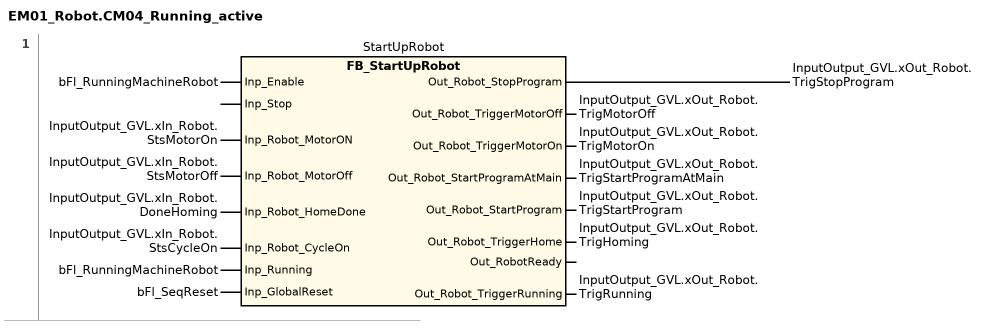
// NETWORK 1
StartUpRobot(
    Inp_Enable := bFl_RunningMachineRobot,
    Inp_Robot_MotorON := InputOutput_GVL.xIn_Robot.StsMotorOn,
    Inp_Robot_MotorOff := InputOutput_GVL.xIn_Robot.StsMotorOff,
    Inp_Robot_HomeDone := InputOutput_GVL.xIn_Robot.DoneHoming,
    Inp_Robot_CycleOn := InputOutput_GVL.xIn_Robot.StsCycleOn,
    Inp_Running := bFl_RunningMachineRobot,
    Inp_GlobalReset := bFl_SeqReset,
    Out_Robot_TriggerMotorOff => InputOutput_GVL.xOut_Robot.TrigMotorOff,
    Out_Robot_TriggerMotorOn => InputOutput_GVL.xOut_Robot.TrigMotorOn,
    Out_Robot_StartProgramAtMain => InputOutput_GVL.xOut_Robot.TrigStartProgramAtMain,
    Out_Robot_StartProgram => InputOutput_GVL.xOut_Robot.TrigStartProgram,
    Out_Robot_TriggerHome => InputOutput_GVL.xOut_Robot.TrigHoming,
    Out_Robot_TriggerRunning => InputOutput_GVL.xOut_Robot.TrigRunning); // FB_StartUpRobot
InputOutput_GVL.xOut_Robot.TrigStopProgram := StartUpRobot.Out_Robot_StopProgram;
END_ACTION

ACTION UP01_Backbone_active:
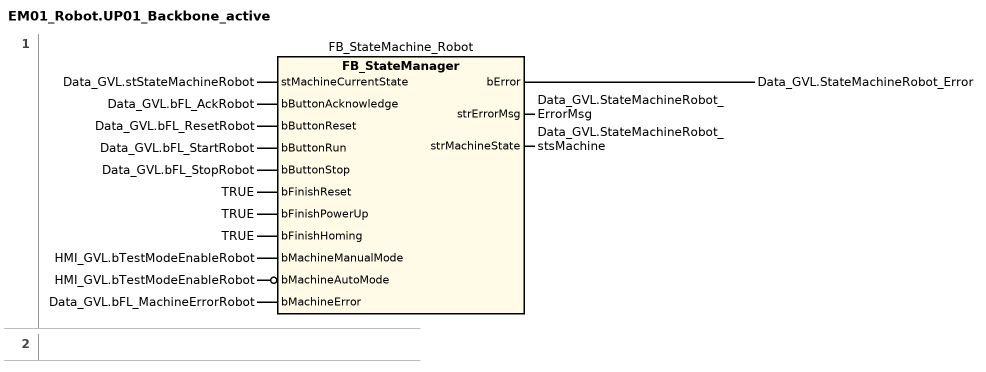
// NETWORK 1
FB_StateMachine_Robot(
    stMachineCurrentState := Data_GVL.stStateMachineRobot,
    bButtonAcknowledge := Data_GVL.bFL_AckRobot,
    bButtonReset := Data_GVL.bFL_ResetRobot,
    bButtonRun := Data_GVL.bFL_StartRobot,
    bButtonStop := Data_GVL.bFL_StopRobot,
    bFinishReset := TRUE,
    bFinishPowerUp := TRUE,
    bFinishHoming := TRUE,
    bMachineManualMode := HMI_GVL.bTestModeEnableRobot,
    bMachineAutoMode := NOT HMI_GVL.bTestModeEnableRobot,
    bMachineError := Data_GVL.bFL_MachineErrorRobot,
    strErrorMsg => Data_GVL.StateMachineRobot_ErrorMsg,
    strMachineState => Data_GVL.StateMachineRobot_stsMachine); // FB_StateManager
Data_GVL.StateMachineRobot_Error := FB_StateMachine_Robot.bError;

// NETWORK 2
END_ACTION

END_PROGRAM

// ---- POUs/Function_Block/General/FB_StateManager.TcPOU
FUNCTION_BLOCK FB_StateManager
VAR_IN_OUT
	stMachineCurrentState			: stMachineState;
END_VAR
VAR_INPUT
	bButtonAcknowledge				: BOOL;		// User Input for Error Acknowledgement
	bButtonReset					: BOOL;		// User Input for Reset 
	bButtonRun						: BOOL;		// User Input for Starting Machine Running Sequence
	bButtonStop						: BOOL;		// User Input for Stopping Machine Running Sequence
	bFinishReset					: BOOL;
	bFinishPowerUp					: BOOL;
	bFinishHoming					: BOOL;
	bMachineManualMode				: BOOL;		// Input(s) Required to Change Machine Operation Mode Into Manual Mode
	bMachineAutoMode				: BOOL;		// Input(s) Required to Change Machine Operation Mode Into Auto Mode
	bMachineError					: BOOL;		// Input(s) required to make the machine goes into error state
END_VAR
VAR_OUTPUT
	bError							: BOOL;		
	strErrorMsg						: STRING;	
	strMachineState					: STRING;
END_VAR
VAR
	bFL_AutoModeActive				: BOOL;
	bFL_ManualModeActive			: BOOL;
	bInit							: BOOL;
	StateIndex						: UINT;
	bFL_Error						: BOOL;
	F_TRIG_AUTO						: F_TRIG;
	F_TRIG_MANUAL					: F_TRIG;
END_VAR

//=======StateManager v1.1=======
//Used UDTs: MachineState - v1.0
//
//Changelog: 
//v1.1 [23.02.2022] Edit Mode selection logic - Fabrilian Asali
//v1.0 [15.01.2021] Start Function block development - Fabrilian Asali
//
//===================================

// Inisialisasi state mesin saat program pertama kali dijalankan
IF NOT bInit THEN
    stMachineCurrentState.Error       := FALSE;          // Set error state mesin menjadi false
    stMachineCurrentState.CheckSafety := FALSE;          // Set status pemeriksaan keselamatan menjadi false
    stMachineCurrentState.Aborted     := FALSE;          // Set status pembatalan menjadi false
    stMachineCurrentState.Initialize  := FALSE;          // Set status inisialisasi menjadi false
    stMachineCurrentState.CheckToRun  := FALSE;          // Set status pemeriksaan untuk menjalankan menjadi false
    stMachineCurrentState.Ready       := FALSE;          // Set status siap menjadi false
    stMachineCurrentState.Running     := FALSE;          // Set status berjalan menjadi false
    stMachineCurrentState.Stopped     := FALSE;          // Set status berhenti menjadi false
    stMachineCurrentState.ManualMode  := FALSE;          // Set status mode manual menjadi false
    bFL_Error  := FALSE;                                 // Set flag error menjadi false
    StateIndex := 0;                                     // Set indeks state menjadi 0
    bInit      := TRUE;                                  // Set flag inisialisasi menjadi true
END_IF;

// Logika untuk mendeteksi kesalahan dan mengatur status mesin menjadi kesalahan jika terdeteksi
IF bMachineError AND NOT bFL_Error THEN
    StateIndex := 0;                 // Set indeks state menjadi 0
    bFL_Error  := TRUE;              // Set flag error menjadi true
END_IF;

// Logika untuk mereset pesan kesalahan saat tombol acknowledge ditekan
IF bButtonAcknowledge THEN
    bError      := FALSE;                // Set status error menjadi false
    strErrorMsg := '';                   // Kosongkan pesan kesalahan
END_IF;

// Logika pemilihan mode otomatis/manual
IF bMachineAutoMode AND NOT bMachineManualMode THEN  //jika status mode aktif & mode mesin manual non-aktif, maka
    bFL_AutoModeActive   := TRUE;      // Set flag mode otomatis aktif menjadi true
    bFL_ManualModeActive := FALSE;     // Set flag mode manual aktif menjadi false
ELSIF NOT bMachineAutoMode AND bMachineManualMode THEN
    bFL_AutoModeActive   := FALSE;       // Set flag mode otomatis aktif menjadi false
    bFL_ManualModeActive := TRUE;        // Set flag mode manual aktif menjadi true
ELSE
    bError               := TRUE;                               // Set status error menjadi true
    strErrorMsg          := 'Operation Mode Fault Detected.';   // Set pesan kesalahan
    bFL_AutoModeActive   := FALSE;                              // Set flag mode otomatis aktif menjadi false
    bFL_ManualModeActive := FALSE;                              // Set flag mode manual aktif menjadi false
END_IF;

// Trigger untuk deteksi perubahan mode otomatis
F_TRIG_AUTO(CLK := bMachineAutoMode);
// Trigger untuk deteksi perubahan mode manual
F_TRIG_MANUAL(CLK := bMachineManualMode);
// Logika untuk menangani perubahan mode otomatis atau manual
IF F_TRIG_AUTO.Q OR F_TRIG_MANUAL.Q THEN
    bError := TRUE;                                     // Set status error menjadi true
    strErrorMsg := 'Operation Mode Change Detected.';   // Set pesan kesalahan
    bFL_AutoModeActive := FALSE;                        // Set flag mode otomatis aktif menjadi false
    bFL_ManualModeActive := FALSE;                      // Set flag mode manual aktif menjadi false
    StateIndex := 0;                                    // Set indeks state menjadi 0
END_IF

	
	
	//V1.0 Selection Logic Code
	
		(*
		IF bMachineAutoMode AND NOT bMachineManualMode THEN
			bFL_AutoModeActive 							:= TRUE;
			bFL_ManualModeActive					 	:= FALSE;
		ELSIF NOT bMachineAutoMode AND bMachineManualMode THEN
			bFL_ManualModeActive					 	:= TRUE;
			bFL_AutoModeActive 							:= FALSE;
		ELSE
			bError 										:= TRUE;
			strErrorMsg 								:= 'Operation Mode Change Detected.';
			bFL_AutoModeActive 							:= FALSE;
			bFL_ManualModeActive						:= FALSE;
		END_IF;
		*)




CASE StateIndex OF
	0: //Error State
		stMachineCurrentState.Error 		:= TRUE;
		stMachineCurrentState.CheckSafety	:= FALSE;
		stMachineCurrentState.Aborted		:= FALSE;
		stMachineCurrentState.Initialize	:= FALSE;
		stMachineCurrentState.CheckToRun	:= FALSE;
		stMachineCurrentState.Ready			:= FALSE;
		stMachineCurrentState.Running		:= FALSE;
		stMachineCurrentState.Stopped		:= FALSE;
		stMachineCurrentState.ManualMode	:= FALSE;
		strMachineState						:= 'Error';
		IF bButtonAcknowledge THEN		
			StateIndex := 10;
		END_IF;
	
	10: //CheckSafety State
		stMachineCurrentState.Error 		:= FALSE;
		stMachineCurrentState.CheckSafety	:= TRUE;
		stMachineCurrentState.Aborted		:= FALSE;
		stMachineCurrentState.Initialize	:= FALSE;
		stMachineCurrentState.CheckToRun	:= FALSE;
		stMachineCurrentState.Ready			:= FALSE;
		stMachineCurrentState.Running		:= FALSE;
		stMachineCurrentState.Stopped		:= FALSE;
		stMachineCurrentState.ManualMode	:= FALSE;
		strMachineState						:= 'Safety';
		IF NOT bMachineError THEN		
			StateIndex 	:= 20;
			bFL_Error		:= FALSE;
		ELSE
			bError 			:= TRUE;
			strErrorMsg := 'Machine Check Safety Failed';
			StateIndex	:= 0;
		END_IF;	

	20: //Aborted State | auto manual mode branching
		stMachineCurrentState.Error 		:= FALSE;
		stMachineCurrentState.CheckSafety	:= FALSE;
		stMachineCurrentState.Aborted		:= TRUE;
		stMachineCurrentState.Initialize	:= FALSE;
		stMachineCurrentState.CheckToRun	:= FALSE;
		stMachineCurrentState.Ready			:= FALSE;
		stMachineCurrentState.Running		:= FALSE;
		stMachineCurrentState.Stopped		:= FALSE;
		stMachineCurrentState.ManualMode	:= FALSE;
		strMachineState						:= 'Aborted';		
		IF bFL_AutoModeActive AND bButtonReset THEN
			StateIndex := 30;
		ELSIF bFL_ManualModeActive THEN
			StateIndex := 1000;
		END_IF;

	30: //Initialize State
		stMachineCurrentState.Error 		:= FALSE;
		stMachineCurrentState.CheckSafety	:= FALSE;
		stMachineCurrentState.Aborted		:= FALSE;
		stMachineCurrentState.Initialize	:= TRUE;
		stMachineCurrentState.CheckToRun	:= FALSE;
		stMachineCurrentState.Ready			:= FALSE;
		stMachineCurrentState.Running		:= FALSE;
		stMachineCurrentState.Stopped		:= FALSE;
		stMachineCurrentState.ManualMode	:= FALSE;
		strMachineState						:= 'Initialize';				
		IF bFinishReset AND bFinishPowerUp THEN
			StateIndex := 40;
		END_IF;
		
	40: //CheckToRun State
		stMachineCurrentState.Error 		:= FALSE;
		stMachineCurrentState.CheckSafety	:= FALSE;
		stMachineCurrentState.Aborted		:= FALSE;
		stMachineCurrentState.Initialize	:= FALSE;
		stMachineCurrentState.CheckToRun	:= TRUE;
		stMachineCurrentState.Ready			:= FALSE;
		stMachineCurrentState.Running		:= FALSE;
		stMachineCurrentState.Stopped		:= FALSE;
		stMachineCurrentState.ManualMode	:= FALSE;
		strMachineState						:= 'Check Run';		
		IF bFinishHoming THEN
			StateIndex := 50;
		END_IF;
		
	50: //Ready State
		stMachineCurrentState.Error 		:= FALSE;
		stMachineCurrentState.CheckSafety	:= FALSE;
		stMachineCurrentState.Aborted		:= FALSE;
		stMachineCurrentState.Initialize	:= FALSE;
		stMachineCurrentState.CheckToRun	:= FALSE;
		stMachineCurrentState.Ready			:= TRUE;
		stMachineCurrentState.Running		:= FALSE;
		stMachineCurrentState.Stopped		:= FALSE;
		stMachineCurrentState.ManualMode	:= FALSE;
		strMachineState						:= 'Ready';				
		IF bButtonRun THEN
			StateIndex := 60;
		END_IF;
		
	60: //Running State
		stMachineCurrentState.Error 		:= FALSE;
		stMachineCurrentState.CheckSafety	:= FALSE;
		stMachineCurrentState.Aborted		:= FALSE;
		stMachineCurrentState.Initialize	:= FALSE;
		stMachineCurrentState.CheckToRun	:= FALSE;
		stMachineCurrentState.Ready			:= FALSE;
		stMachineCurrentState.Running		:= TRUE;
		stMachineCurrentState.Stopped		:= FALSE;
		stMachineCurrentState.ManualMode	:= FALSE;
		strMachineState						:= 'Running';		
		IF bButtonStop THEN
			StateIndex := 70;
		END_IF;
		
	70: //Stopped State
		stMachineCurrentState.Error 		:= FALSE;
		stMachineCurrentState.CheckSafety	:= FALSE;
		stMachineCurrentState.Aborted		:= FALSE;
		stMachineCurrentState.Initialize	:= FALSE;
		stMachineCurrentState.CheckToRun	:= FALSE;
		stMachineCurrentState.Ready			:= FALSE;
		stMachineCurrentState.Running		:= FALSE;
		stMachineCurrentState.Stopped		:= TRUE;
		stMachineCurrentState.ManualMode	:= FALSE;
		strMachineState						:= 'Stopped';
		IF bButtonRun THEN
			StateIndex := 60;
		END_IF;
		
	1000: //Manual mode operation state
		stMachineCurrentState.Error 		:= FALSE;
		stMachineCurrentState.CheckSafety	:= FALSE;
		stMachineCurrentState.Aborted		:= FALSE;
		stMachineCurrentState.Initialize	:= FALSE;
		stMachineCurrentState.CheckToRun	:= FALSE;
		stMachineCurrentState.Ready			:= FALSE;
		stMachineCurrentState.Running		:= FALSE;
		stMachineCurrentState.Stopped		:= FALSE;
		stMachineCurrentState.ManualMode	:= TRUE;
		strMachineState						:= 'Manual';
		IF bFL_AutoModeActive THEN
			StateIndex := 0;
		END_IF
END_CASE;

END_FUNCTION_BLOCK

// ---- POUs/Function_Block/General/CheckStatus.TcPOU
FUNCTION_BLOCK CheckStatus
VAR_INPUT
	F_Reset: BOOL;
	Data: ARRAY [1..100] OF BOOL;
END_VAR
VAR_OUTPUT
	Status: BOOL;
	Reset : R_TRIG;
END_VAR
VAR
	i: UINT;
	j: UINT;
	
	a: UINT;
	
	SeqCheck: ARRAY [1..300] OF UINT;
	CheckReset: BOOL;
	SeqIndex: INT;
END_VAR

(* new Management Error *)
CASE SeqIndex OF 
	0: 
		FOR i:=1 TO 100 BY 1 DO //program for ini bertujuan untuk mengiterasi i dari 1 sampai 100
			IF Data[i] THEN		//jika pada iterasi Data terdapat nilai ke-i = true
				Status:=TRUE;   //maka output status menjadi true
				j := 0;         //dan index j = 0
				i := 100;       //dan index i = 100
				seqIndex := 10; //SeqIndex berpindah ke 10
			END_IF
			
		END_FOR
	10: 
		Reset( CLK := F_Reset);               //Raising Trigger/Trigger Positif didapat oleh F_Reset, maka reset akan aktif
		IF Reset.Q AND NOT CheckReset THEN    //jika reset bernilai TRUE dan CheckReset bernilai FALSE, maka:
			i := 0;                           //index = 0
			CheckReset:=TRUE;                 //CheckReset = TRUE
			seqIndex := 20;                   //SeqIndex berpindah ke sequence 20
		END_IF
	20: 
		IF CheckReset THEN 
			FOR j:=1 TO 100 BY 1 DO           //iterasikan j dari 1 sampai dengan 100
				IF NOT Data[j] THEN		      //jika dalam array data J terdapoat nilai TRUE
					Status:=FALSE;            //Status jadi False
					CheckReset:=FALSE;        //CheckReset jadi False
					j := 100 ;                //J berubah index ke 100
					seqIndex := 0;            //SeqIndex berubah ke keadaan awal
				END_IF
			END_FOR
		END_IF 
END_CASE
(* old management error *problem Delay Respons
IF CheckReset THEN
	CASE SeqCheck[a] OF
		0:
			IF NOT Data[a] THEN
				SeqCheck[a]:=10;
			ELSE
				CheckReset:=FALSE;
			END_IF
		10:
			IF a = 300 THEN
				Status:=FALSE;
				CheckReset:=FALSE;
			ELSE
				a := a + 1;
			END_IF
	END_CASE
ELSE
	FOR j:=1 TO 300 BY 1 DO
		SeqCheck[j]:=0;
	END_FOR
	a:=1;
END_IF

*)

END_FUNCTION_BLOCK

// ---- POUs/Function_Block/Robot/FB_StartUpRobot.TcPOU
FUNCTION_BLOCK FB_StartUpRobot
VAR_INPUT
	Inp_Enable					: BOOL;
	Inp_Stop					: BOOL;
	Inp_Robot_MotorON			: BOOL;
	Inp_Robot_MotorOff			: BOOL;
	Inp_Robot_HomeDone			: BOOL;
	Inp_Robot_CycleOn			: BOOL;
	Inp_Running					: BOOL;
	Inp_GlobalReset				: BOOL;
END_VAR
VAR_OUTPUT
	Out_Robot_StopProgram		: BOOL;
	Out_Robot_TriggerMotorOff	: BOOL;
	Out_Robot_TriggerMotorOn	: BOOL;
	Out_Robot_StartProgramAtMain: BOOL;
	Out_Robot_StartProgram		: BOOL;
	Out_Robot_TriggerHome		: BOOL;
	Out_RobotReady				: BOOL;
	Out_Robot_TriggerRunning	: BOOL;
END_VAR
VAR
	Sequence_Abort				: INT;
	Sequence_Run				: INT;
	DataTimer					: TON;
	Sts_RobotHasBeenRun			: BOOL;
	Sts_RobotHasBeenHome		: BOOL;
END_VAR

IF Inp_Enable AND NOT Inp_Stop THEN
    
    Sequence_Abort := 0;
    Out_Robot_StopProgram := FALSE;
    Out_Robot_TriggerMotorOff := FALSE;
    
    CASE Sequence_Run OF
        0:
            IF Inp_Robot_MotorOff AND NOT Inp_Robot_MotorON THEN
                Sequence_Run := 10;
            ELSIF NOT Inp_Robot_MotorOff AND Inp_Robot_MotorON THEN
                Sequence_Run := 20;
            END_IF;
        10:
            Out_Robot_TriggerMotorOn := TRUE;
            IF NOT Inp_Robot_MotorOff AND Inp_Robot_MotorON THEN
                Out_Robot_TriggerMotorOn := FALSE;
				DataTimer(IN := FALSE);
                Sequence_Run := 30;
            ELSE
                DataTimer(IN := TRUE,PT := T#100MS);
                IF DataTimer.Q THEN
                    DataTimer(IN := FALSE);
                    Sequence_Run := 0;
                END_IF;
            END_IF;
        20:
            Out_Robot_TriggerMotorOn := FALSE;
            IF NOT Sts_RobotHasBeenRun THEN
                Sequence_Run := 30;
            ELSE
                Sequence_Run := 40;
            END_IF;
        30:
            Out_Robot_StartProgramAtMain := TRUE;
            IF Inp_Robot_CycleOn THEN
                Sts_RobotHasBeenRun := TRUE;
                Out_Robot_StartProgramAtMain := FALSE;
				DataTimer(IN := FALSE);
                Sequence_Run := 50;
            ELSE
                DataTimer(IN := TRUE,PT := T#100MS);
                IF DataTimer.Q THEN
                    DataTimer(IN := FALSE);
                    Sequence_Run := 20;
                END_IF;
            END_IF;
        40:
            Out_Robot_StartProgram := TRUE;
            IF Inp_Robot_CycleOn THEN
                Out_Robot_StartProgram:= FALSE;
				DataTimer(IN := FALSE);
                Sequence_Run := 50;
            ELSE
                DataTimer(IN := TRUE,PT := T#100MS);
                IF DataTimer.Q THEN
                    DataTimer(IN := FALSE);
                    Sequence_Run := 20;
                END_IF;
            END_IF;
        50:
            IF NOT Sts_RobotHasBeenHome THEN
                Sequence_Run := 60;
            ELSE
                Sequence_Run := 80;
            END_IF;
        60:
            Out_Robot_TriggerHome := TRUE;
            IF Inp_Robot_HomeDone THEN
                Out_Robot_TriggerHome := FALSE;
                Sequence_Run := 70;
            END_IF;
        70:
            IF NOT Inp_Robot_HomeDone THEN
                Sts_RobotHasBeenHome:= TRUE;
                Sequence_Run := 80;
            END_IF;
        80:
            Out_RobotReady := TRUE;
            IF Inp_Running THEN
                Sequence_Run := 90;
            END_IF;
        90:
            Out_Robot_TriggerRunning := TRUE;
                
    END_CASE;
    
ELSE
    
    CASE Sequence_Abort OF
        0:
            IF Inp_Robot_CycleOn THEN
                Sequence_Abort := 10;
            ELSE
                Sequence_Abort := 20;
            END_IF;
        10:
            Out_Robot_StopProgram := TRUE;
            IF NOT Inp_Robot_CycleOn THEN
                Out_Robot_StopProgram := FALSE;
				DataTimer(IN := FALSE);
                Sequence_Abort := 20;
            ELSE
                DataTimer(IN := TRUE,PT := T#100MS);
                IF DataTimer.Q THEN
                    DataTimer(IN := FALSE);
                    Out_Robot_StopProgram := FALSE;
                    Sequence_Abort := 0;
                END_IF;
            END_IF;
        20:
            IF Inp_Robot_MotorON AND NOT Inp_Robot_MotorOff THEN
                Sequence_Abort := 25;
            ELSIF NOT Inp_Robot_MotorON AND Inp_Robot_MotorOff THEN
                Sequence_Abort := 40;
            END_IF;
        25:
            DataTimer(IN := TRUE,PT := T#100MS);
                IF DataTimer.Q THEN
                    DataTimer(IN := FALSE);
                    Out_Robot_StopProgram := FALSE;
                    Sequence_Abort := 30;
                END_IF;
        30:
            Out_Robot_TriggerMotorOff := TRUE;
            IF Inp_Robot_MotorOff AND NOT Inp_Robot_MotorON THEN
                Out_Robot_TriggerMotorOff := FALSE;
                Sequence_Abort := 30;
            ELSE
               DataTimer(IN := TRUE,PT := T#100MS);
                IF DataTimer.Q THEN
                    DataTimer(IN := FALSE);
                    Out_Robot_StopProgram := FALSE;
                    Sequence_Abort := 20;
                END_IF;
            END_IF;
			40:
			        Out_Robot_TriggerMotorOff := FALSE;
					
    END_CASE;
    
    DataTimer(IN := FALSE);
    Sequence_Run := 0;
    Out_Robot_TriggerRunning := FALSE;
    Out_Robot_TriggerMotorOn := FALSE;
    Out_Robot_StartProgram := FALSE;
    Out_Robot_StartProgramAtMain := FALSE;
    Out_Robot_TriggerHome := FALSE;
    
    IF Inp_GlobalReset THEN
        Out_RobotReady := FALSE;
        Sts_RobotHasBeenRun := FALSE;
        Sts_RobotHasBeenHome := FALSE;
    END_IF;
	
	IF Inp_Stop THEN
		Out_Robot_StopProgram:=TRUE;
	END_IF;
    
END_IF;

END_FUNCTION_BLOCK

// ---- POUs/S02_Placing/EM02_Placing1.TcPOU
PROGRAM EM02_Placing1
VAR
	
	//Backbone
	FB_StateMachine_Placing1		: FB_StateManager;
	bFl_RunningMachinePlacing1		: BOOL;
	bFl_SeqReset					: BOOL;
	bFl_Manual						: BOOL;
	CheckStatusPlacing1				: checkstatus;
	AlarmEventHistory				: ARRAY[1..20] OF Alarm_Event_History;
	Placing1_Management				: FB_Placing_v2;
	bFl_Flushing					: BOOL;
	PalletID_Placing1				: PalletID_name;
	Placing1_ID						: STRING;
	bFl_PalletJammed				: BOOL;
	
	//Motor
	Motor_PalletPlacing1			: MotorManagement;
	bFl_MotorPlacing1				: BOOL;
	Motor_Placing1_Error			: BOOL;
	Motor_Placing1_ErrorID			: UINT;
	bFl_MotorPlacing1_Fwd			: BOOL;
	bFl_MotorPlacing1_Rev			: BOOL;
	bFL_Safety						: BOOL;
	AlarmEventActive				: ARRAY[1..20] OF Alarm_Event_Active;
	CheckAcc						: TON;
END_VAR
VAR // added by the converter: edge detectors and wires of the graphical bodies
    _w1 : BOOL;
END_VAR

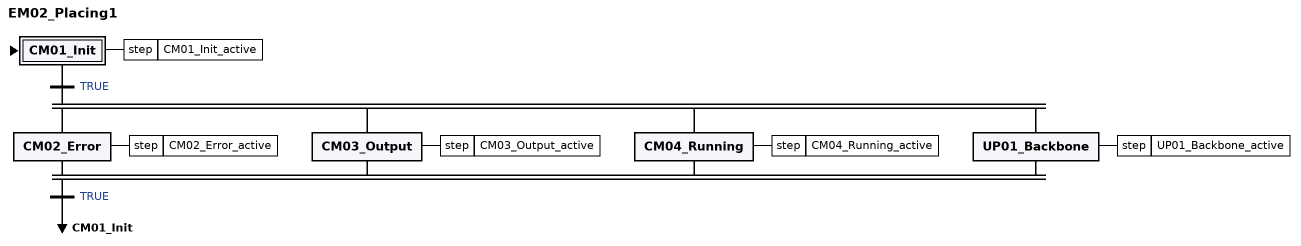
INITIAL_STEP CM01_Init:
    CM01_Init_active(N);  // step action
END_STEP
TRANSITION FROM CM01_Init TO (CM02_Error, CM03_Output, CM04_Running, UP01_Backbone)
    := TRUE;
END_TRANSITION
STEP CM02_Error:
    CM02_Error_active(N);  // step action
END_STEP
STEP CM03_Output:
    CM03_Output_active(N);  // step action
END_STEP
STEP CM04_Running:
    CM04_Running_active(N);  // step action
END_STEP
STEP UP01_Backbone:
    UP01_Backbone_active(N);  // step action
END_STEP
TRANSITION FROM (CM02_Error, CM03_Output, CM04_Running, UP01_Backbone) TO CM01_Init
    := TRUE;
END_TRANSITION

ACTION CM01_Init_active:
Data_GVL.bFL_StartPlacing1			:= Status_GVL.bFl_RunButton_Robotic OR HMI_GVL.bStartButtonPlacing1;
Data_GVL.bFL_StopPlacing1			:= NOT Status_GVL.bFl_StopButton_Robotic OR HMI_GVL.bStopButtonPlacing1;
Data_GVL.bFL_ResetPlacing1			:= Status_GVL.bFl_ResetButton_Robotic OR HMI_GVL.bResetButtonPlacing1;
Data_GVL.bFL_AckPlacing1			:= Status_GVL.bFl_Acknowledge_Robotic OR HMI_GVL.bAcknowledgeButtonPlacing1;
Data_GVL.bFL_AutoManuaModePlacing1 	:= Status_GVL.bFl_Manual_Robotic OR HMI_GVL.bTestModeEnablePlacing1;
bFl_RunningMachinePlacing1			:= Data_GVL.stStateMachinePlacing1.Running;
bFl_Manual							:= Data_GVL.stStateMachinePlacing1.ManualMode;
bFl_SeqReset						:= NOT Status_GVL.bFl_EStop_Robotic;
bFL_Safety							:= Status_GVL.bFl_EStop_Robotic AND Status_GVL.bSafety_DoorRobotic;


(*=================Convert Timer============================*)
Data_GVL.Tmr_Placing1	:= ConvertMilliSecTimeData(HMI_GVL.Tmr_Placing1);

(*=================Data OEE============================*)
Data_GVL.dt_Production[1].Data1			:= HMI_GVL.arCountTotal[1];
Data_GVL.dt_Production[1].Data2			:= HMI_GVL.arPalletTotal[1];
Data_GVL.dt_Production[1].Data3			:= HMI_GVL.arPalletIncomplete[1];
Data_GVL.dt_Production[1].ProductCode	:= Status_GVL.RecipeLine[1].ProductName;
END_ACTION

ACTION CM02_Error_active:
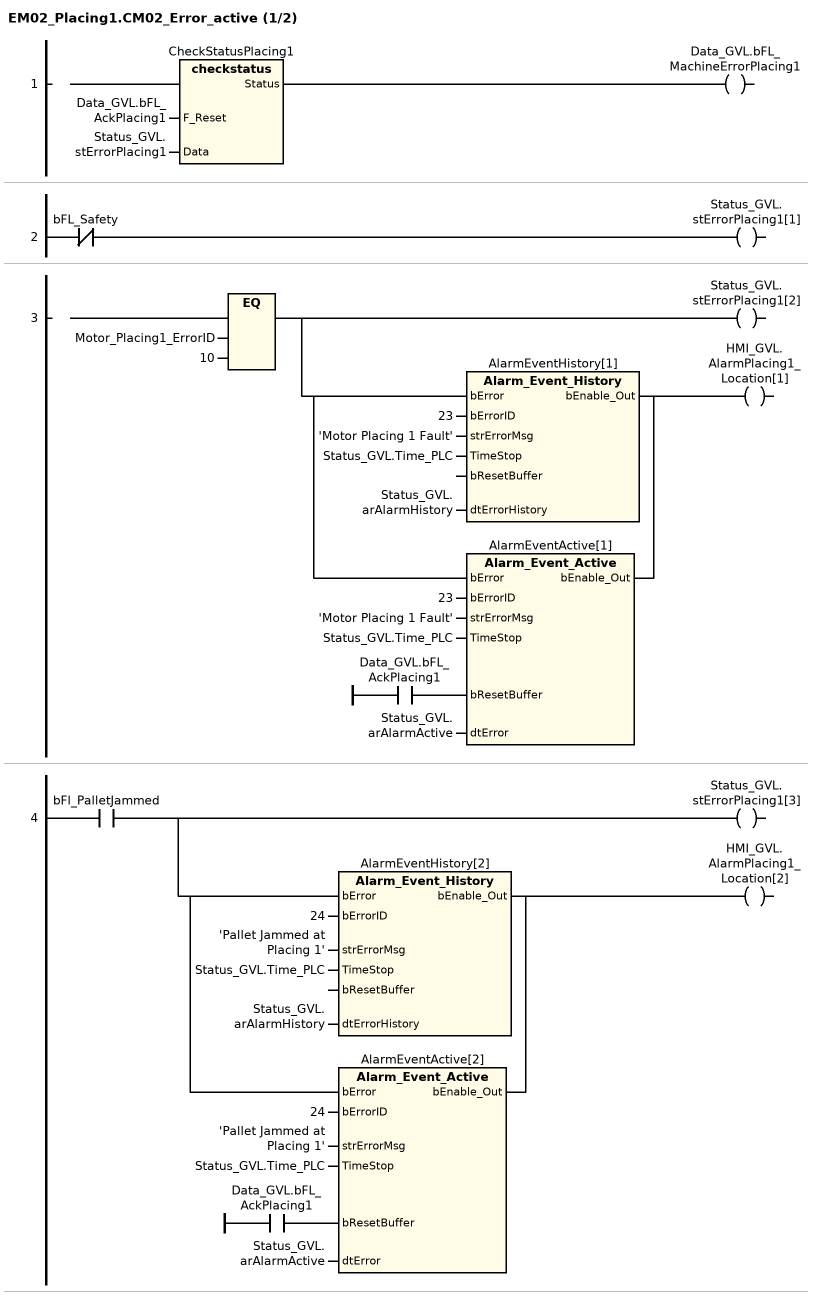
// NETWORK 1
CheckStatusPlacing1(F_Reset := Data_GVL.bFL_AckPlacing1, Data := Status_GVL.stErrorPlacing1); // checkstatus
Data_GVL.bFL_MachineErrorPlacing1 := CheckStatusPlacing1.Status;

// NETWORK 2
Status_GVL.stErrorPlacing1[1] := NOT bFL_Safety;

// NETWORK 3
_w1 := Motor_Placing1_ErrorID = 10;
Status_GVL.stErrorPlacing1[2] := _w1;
AlarmEventHistory[1](
    bError := _w1,
    bErrorID := 23,
    strErrorMsg := 'Motor Placing 1 Fault',
    TimeStop := Status_GVL.Time_PLC,
    dtErrorHistory := Status_GVL.arAlarmHistory); // Alarm_Event_History
AlarmEventActive[1](
    bError := _w1,
    bErrorID := 23,
    strErrorMsg := 'Motor Placing 1 Fault',
    TimeStop := Status_GVL.Time_PLC,
    bResetBuffer := Data_GVL.bFL_AckPlacing1,
    dtError := Status_GVL.arAlarmActive); // Alarm_Event_Active
HMI_GVL.AlarmPlacing1_Location[1] := AlarmEventHistory[1].bEnable_Out OR AlarmEventActive[1].bEnable_Out;

// NETWORK 4
Status_GVL.stErrorPlacing1[3] := bFl_PalletJammed;
AlarmEventHistory[2](
    bError := bFl_PalletJammed,
    bErrorID := 24,
    strErrorMsg := 'Pallet Jammed at Placing 1',
    TimeStop := Status_GVL.Time_PLC,
    dtErrorHistory := Status_GVL.arAlarmHistory); // Alarm_Event_History
AlarmEventActive[2](
    bError := bFl_PalletJammed,
    bErrorID := 24,
    strErrorMsg := 'Pallet Jammed at Placing 1',
    TimeStop := Status_GVL.Time_PLC,
    bResetBuffer := Data_GVL.bFL_AckPlacing1,
    dtError := Status_GVL.arAlarmActive); // Alarm_Event_Active
HMI_GVL.AlarmPlacing1_Location[2] := AlarmEventHistory[2].bEnable_Out OR AlarmEventActive[2].bEnable_Out;

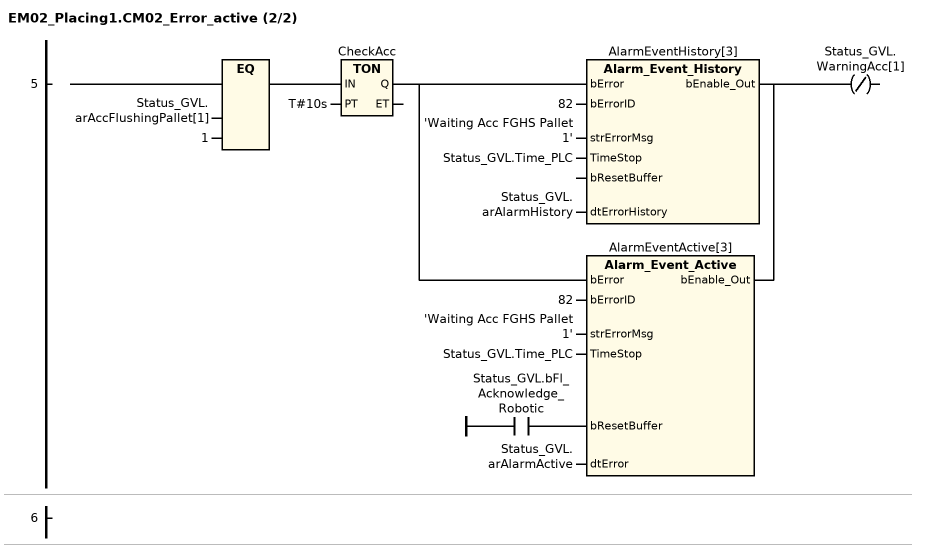
// NETWORK 5
CheckAcc(IN := Status_GVL.arAccFlushingPallet[1] = 1, PT := T#10s); // TON
AlarmEventHistory[3](
    bError := CheckAcc.Q,
    bErrorID := 82,
    strErrorMsg := 'Waiting Acc FGHS Pallet 1',
    TimeStop := Status_GVL.Time_PLC,
    dtErrorHistory := Status_GVL.arAlarmHistory); // Alarm_Event_History
AlarmEventActive[3](
    bError := CheckAcc.Q,
    bErrorID := 82,
    strErrorMsg := 'Waiting Acc FGHS Pallet 1',
    TimeStop := Status_GVL.Time_PLC,
    bResetBuffer := Status_GVL.bFl_Acknowledge_Robotic,
    dtError := Status_GVL.arAlarmActive); // Alarm_Event_Active
Status_GVL.WarningAcc[1] := NOT (AlarmEventHistory[3].bEnable_Out OR AlarmEventActive[3].bEnable_Out);

// NETWORK 6
END_ACTION

ACTION CM03_Output_active:
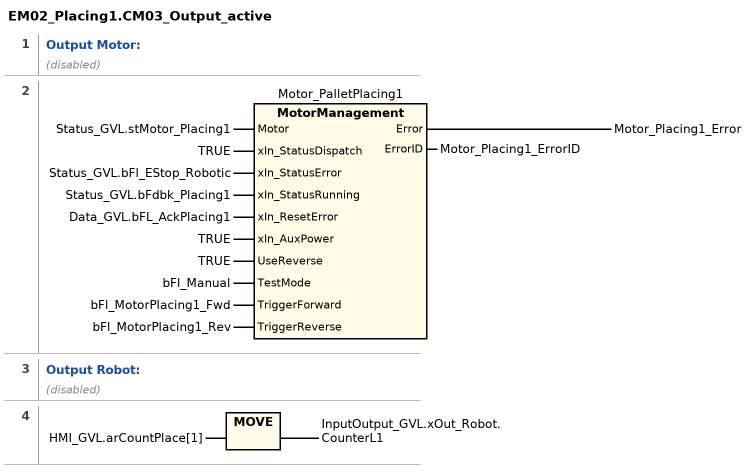
// NETWORK 1 (disabled)
// label: Output Motor

// NETWORK 2
Motor_PalletPlacing1(
    Motor := Status_GVL.stMotor_Placing1,
    xIn_StatusDispatch := TRUE,
    xIn_StatusError := Status_GVL.bFl_EStop_Robotic,
    xIn_StatusRunning := Status_GVL.bFdbk_Placing1,
    xIn_ResetError := Data_GVL.bFL_AckPlacing1,
    xIn_AuxPower := TRUE,
    UseReverse := TRUE,
    TestMode := bFl_Manual,
    TriggerForward := bFl_MotorPlacing1_Fwd,
    TriggerReverse := bFl_MotorPlacing1_Rev,
    ErrorID => Motor_Placing1_ErrorID); // MotorManagement
Motor_Placing1_Error := Motor_PalletPlacing1.Error;

// NETWORK 3 (disabled)
// label: Output Robot

// NETWORK 4
InputOutput_GVL.xOut_Robot.CounterL1 := HMI_GVL.arCountPlace[1];
END_ACTION

ACTION CM04_Running_active:
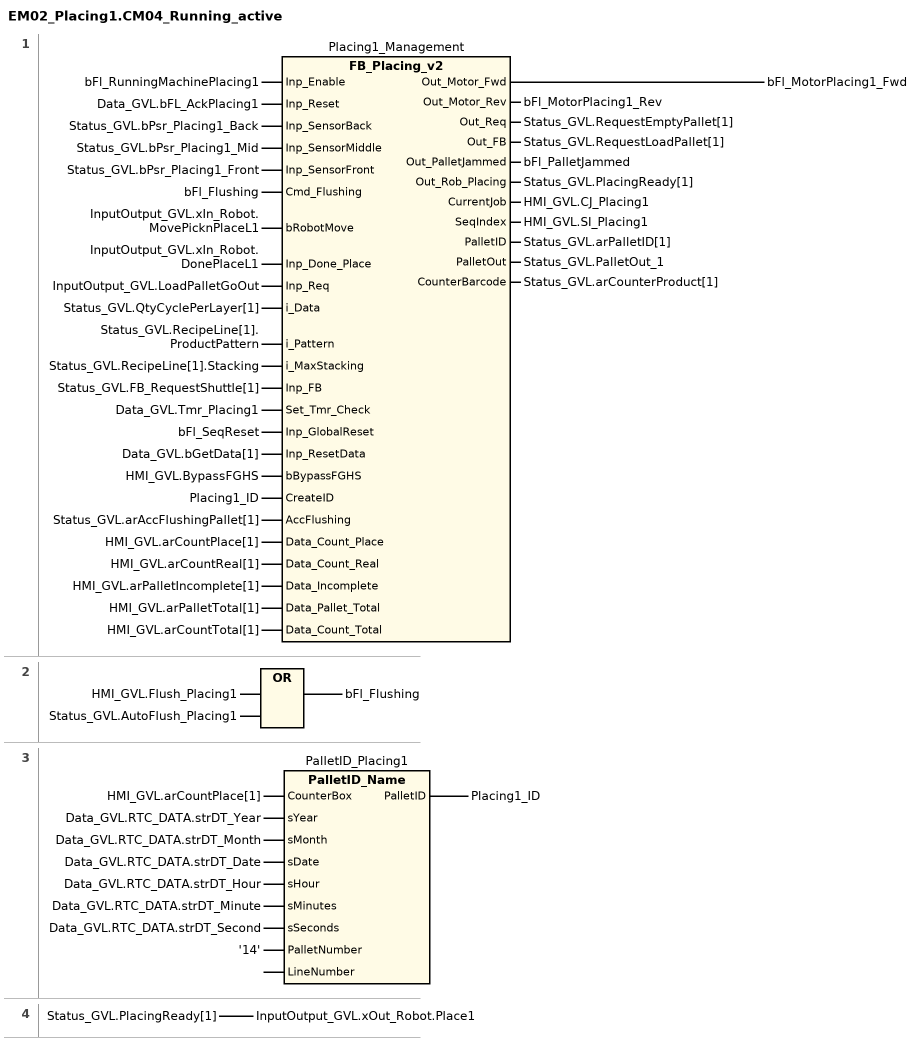
// NETWORK 1
Placing1_Management(
    Inp_Enable := bFl_RunningMachinePlacing1,
    Inp_Reset := Data_GVL.bFL_AckPlacing1,
    Inp_SensorBack := Status_GVL.bPsr_Placing1_Back,
    Inp_SensorMiddle := Status_GVL.bPsr_Placing1_Mid,
    Inp_SensorFront := Status_GVL.bPsr_Placing1_Front,
    Cmd_Flushing := bFl_Flushing,
    bRobotMove := InputOutput_GVL.xIn_Robot.MovePicknPlaceL1,
    Inp_Done_Place := InputOutput_GVL.xIn_Robot.DonePlaceL1,
    Inp_Req := InputOutput_GVL.LoadPalletGoOut,
    i_Data := Status_GVL.QtyCyclePerLayer[1],
    i_Pattern := Status_GVL.RecipeLine[1].ProductPattern,
    i_MaxStacking := Status_GVL.RecipeLine[1].Stacking,
    Inp_FB := Status_GVL.FB_RequestShuttle[1],
    Set_Tmr_Check := Data_GVL.Tmr_Placing1,
    Inp_GlobalReset := bFl_SeqReset,
    Inp_ResetData := Data_GVL.bGetData[1],
    bBypassFGHS := HMI_GVL.BypassFGHS,
    CreateID := Placing1_ID,
    AccFlushing := Status_GVL.arAccFlushingPallet[1],
    Data_Count_Place := HMI_GVL.arCountPlace[1],
    Data_Count_Real := HMI_GVL.arCountReal[1],
    Data_Incomplete := HMI_GVL.arPalletIncomplete[1],
    Data_Pallet_Total := HMI_GVL.arPalletTotal[1],
    Data_Count_Total := HMI_GVL.arCountTotal[1],
    Out_Motor_Rev => bFl_MotorPlacing1_Rev,
    Out_Req => Status_GVL.RequestEmptyPallet[1],
    Out_FB => Status_GVL.RequestLoadPallet[1],
    Out_PalletJammed => bFl_PalletJammed,
    Out_Rob_Placing => Status_GVL.PlacingReady[1],
    CurrentJob => HMI_GVL.CJ_Placing1,
    SeqIndex => HMI_GVL.SI_Placing1,
    PalletID => Status_GVL.arPalletID[1],
    PalletOut => Status_GVL.PalletOut_1,
    CounterBarcode => Status_GVL.arCounterProduct[1]); // FB_Placing_v2
bFl_MotorPlacing1_Fwd := Placing1_Management.Out_Motor_Fwd;

// NETWORK 2
bFl_Flushing := HMI_GVL.Flush_Placing1 OR Status_GVL.AutoFlush_Placing1;

// NETWORK 3
PalletID_Placing1(
    CounterBox := HMI_GVL.arCountPlace[1],
    sYear := Data_GVL.RTC_DATA.strDT_Year,
    sMonth := Data_GVL.RTC_DATA.strDT_Month,
    sDate := Data_GVL.RTC_DATA.strDT_Date,
    sHour := Data_GVL.RTC_DATA.strDT_Hour,
    sMinutes := Data_GVL.RTC_DATA.strDT_Minute,
    sSeconds := Data_GVL.RTC_DATA.strDT_Second,
    PalletNumber := '14'); // PalletID_Name
Placing1_ID := PalletID_Placing1.PalletID;

// NETWORK 4
InputOutput_GVL.xOut_Robot.Place1 := Status_GVL.PlacingReady[1];
END_ACTION

ACTION UP01_Backbone_active:
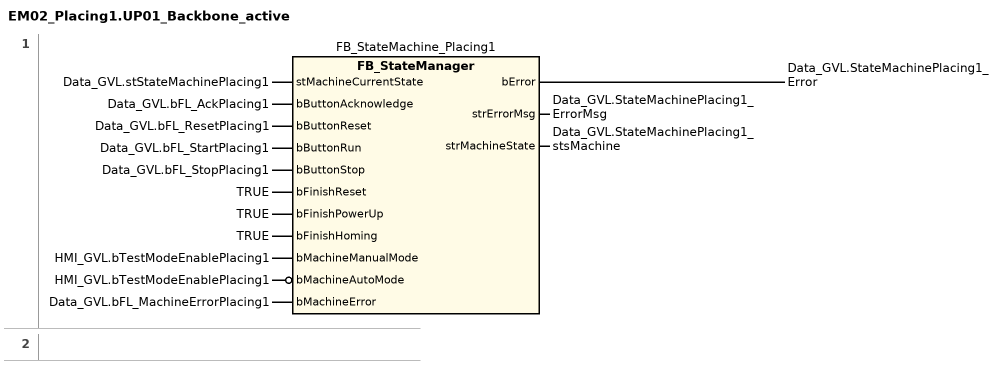
// NETWORK 1
FB_StateMachine_Placing1(
    stMachineCurrentState := Data_GVL.stStateMachinePlacing1,
    bButtonAcknowledge := Data_GVL.bFL_AckPlacing1,
    bButtonReset := Data_GVL.bFL_ResetPlacing1,
    bButtonRun := Data_GVL.bFL_StartPlacing1,
    bButtonStop := Data_GVL.bFL_StopPlacing1,
    bFinishReset := TRUE,
    bFinishPowerUp := TRUE,
    bFinishHoming := TRUE,
    bMachineManualMode := HMI_GVL.bTestModeEnablePlacing1,
    bMachineAutoMode := NOT HMI_GVL.bTestModeEnablePlacing1,
    bMachineError := Data_GVL.bFL_MachineErrorPlacing1,
    strErrorMsg => Data_GVL.StateMachinePlacing1_ErrorMsg,
    strMachineState => Data_GVL.StateMachinePlacing1_stsMachine); // FB_StateManager
Data_GVL.StateMachinePlacing1_Error := FB_StateMachine_Placing1.bError;

// NETWORK 2
END_ACTION

END_PROGRAM

// ---- POUs/Function_Block/Placing/FB_Placing_v2.TcPOU
FUNCTION_BLOCK FB_Placing_v2
VAR_INPUT
	Inp_Enable				: BOOL;
	Inp_Reset				: BOOL;
	Inp_SensorBack			: BOOL;
	Inp_SensorMiddle		: BOOL;
	Inp_SensorFront			: BOOL;
	Cmd_Flushing			: BOOL;
	bRobotMove				: BOOL;
	Inp_Done_Place			: BOOL;
	Inp_Req					: BOOL;
	i_Data					: UINT;
	i_Pattern				: UINT;
	i_MaxStacking			: UINT;
	Inp_FB					: BOOL;
	Set_Tmr_Check			: TIME;
	Inp_GlobalReset			: BOOL;
	Inp_ResetData			: BOOL;
	bBypassFGHS				: BOOL;
	CreateID				: STRING;
	
END_VAR
VAR_OUTPUT
	Out_Motor_Fwd			: BOOL;
	Out_Motor_Rev			: BOOL;
	Out_Req					: BOOL;
	Out_FB					: BOOL;
	Out_PalletJammed		: BOOL;
	Out_Rob_Placing			: BOOL;
	CurrentJob				: STRING;
	SeqIndex				: INT;
	PalletOut				: BOOL;
END_VAR
VAR_OUTPUT PERSISTENT
	PalletID				: STRING;
	CounterBarcode			: BYTE;
END_VAR

VAR
	Sts_Flushing			: BOOL;
	o_MaxCycle				: UINT;
	DataTimer				: TON;
	TWatchDog				: TON;
	Sequence				: INT;
END_VAR

VAR_IN_OUT
	AccFlushing				: BYTE;
	Data_Count_Place		: USINT;
	Data_Count_Real			: USINT;
	Data_Incomplete			: UINT;
	Data_Pallet_Total		: UINT;
	Data_Count_Total		: UINT;
END_VAR

IF Inp_Reset AND Out_PalletJammed THEN
	Out_PalletJammed	:= FALSE;
	Sequence 			:= 0;
END_IF

IF Inp_Enable THEN
	
	IF Cmd_Flushing THEN
		Sts_Flushing:=TRUE;
	END_IF;
	
    CASE Sequence OF
        0:	(* Check Motor *)
			 Out_Motor_Fwd := TRUE;
			 DataTimer(IN:=TRUE, PT:=T#4S);
			 IF DataTimer.Q OR AccFlushing = 2 THEN
				 DataTimer(IN:=FALSE);
				 Out_Motor_Fwd	:= FALSE;
				 Sequence		:= 10;
			 END_IF

		10:  (* Check Sensor *)
			CurrentJob		:= 'Check Sensor';
			IF (Inp_SensorFront OR Inp_SensorMiddle OR Inp_SensorBack) AND AccFlushing = 2 THEN
				Sequence := 600;
			ELSIF (Inp_SensorFront OR Inp_SensorMiddle OR Inp_SensorBack) AND ((Data_Count_Place > o_MaxCycle AND o_MaxCycle <> 0)  OR Sts_Flushing) THEN
                Sequence := 500;
            ELSIF Inp_SensorFront THEN
                Sequence := 300;
            ELSIF NOT Inp_SensorFront AND (Inp_SensorMiddle OR Inp_SensorBack)  THEN
                Sequence := 200;
            ELSE
                Sequence := 100;
            END_IF;
			
			
        100:    (* Request *)
			CurrentJob		:= 'Request Pallet';
			Sts_Flushing	:= FALSE;
            Out_Req			:= TRUE;
			Out_FB			:= FALSE;
            IF Inp_FB THEN
				DataTimer(IN:=FALSE);
                Sequence := 200;
            END_IF;       
			
        200:    (* Pallet Masuk *)
			CurrentJob	:= 'Pallet In';
			PalletOut	:= FALSE;
			IF NOT Inp_SensorFront AND NOT Inp_SensorMiddle AND NOT Inp_SensorBack THEN
            	Out_Req := TRUE;
			END_IF
            Out_Motor_Fwd := TRUE;
            IF Inp_SensorFront AND (Inp_SensorBack OR Inp_SensorMiddle)  THEN
				DataTimer(IN := TRUE,PT := Set_Tmr_Check);
                IF DataTimer.Q THEN
					TWatchDog(IN := FALSE);
                    DataTimer(IN:=FALSE);
					Out_PalletJammed	:= FALSE;
					Out_Motor_Fwd		:= FALSE;
           			Out_Req				:= FALSE;
                    Sequence			:= 300;
                END_IF;    
			ELSE
				TWatchDog(IN := TRUE, PT := T#15S);
				IF TWatchDog.Q THEN
					Sequence	:= 9999;
				END_IF;
            END_IF;
			
        300:
			CurrentJob	:= 'Check Cycle';
			IF o_MaxCycle <> 0 THEN
				IF o_MaxCycle >= Data_Count_Place  THEN
					Sequence := 400;
				ELSE
					DataTimer(IN := TRUE,PT := T#2S);
					IF DataTimer.Q THEN
						DataTimer(IN:=FALSE);
						Sequence := 500;
					END_IF;
				END_IF;
			END_IF
			
        400:
			CurrentJob		:= 'Place Ready';
			AccFlushing		:= 0;
            Out_Rob_Placing := TRUE;
			PalletID			:= CreateID;
            IF Inp_Done_Place THEN
                    Data_Count_Real		:= Data_Count_Real + 1;
                    Data_Count_Place	:= Data_Count_Place + 1;
                    Sequence 			:= 450;
            ELSIF (Cmd_Flushing OR Sts_Flushing) AND NOT bRobotMove THEN
                Data_Incomplete			:= Data_Incomplete + 1;
                Sts_Flushing			:= TRUE;
                Sequence 				:= 500;				
            END_IF;
			
        450:
            Out_Rob_Placing := FALSE;
            IF NOT Inp_Done_Place THEN
                Sequence := 460;
            END_IF;	
			
		460:
			IF PalletID <> '' THEN
				CounterBarcode	:= Data_Count_Real;
				Sequence 		:= 300;
			END_IF
			
		500:
			CurrentJob		:= 'Create Pallet ID';
			DataTimer(IN := TRUE,PT := T#500MS);
			IF DataTimer.Q THEN
				DataTimer(IN := FALSE);
				Sequence		:= 550;
			END_IF
						
		550:
			AccFlushing		:= 1;
			Sequence		:= 600;
			
		600:
			Out_Rob_Placing := FALSE;
			Out_FB 			:= FALSE;
			Out_Req 		:= FALSE;
			CurrentJob		:= 'Waiting Acc Flushing';
			IF (PalletID <> '' AND AccFlushing = 2) OR bBypassFGHS OR Data_Count_Real = 0 THEN
                Sequence := 900;
            END_IF;
		
		900:	(* Positioning Pallet Out *)
			CurrentJob		:= 'Positioning Pallet Out';
			Out_Rob_Placing := FALSE;
			Out_FB 			:= TRUE;
			Out_Req 		:= TRUE;
			Out_Motor_Rev	:= TRUE;
            IF Inp_SensorBack THEN
                DataTimer(IN := TRUE,PT := T#100MS);
                IF DataTimer.Q THEN
					TWatchDog(IN := FALSE);
					DataTimer(IN:=FALSE);
					Out_Motor_Rev	:= FALSE;
                    Sequence		:= 1000;
                END_IF;
			ELSE
				TWatchDog(IN := TRUE, PT := T#15S);
				IF TWatchDog.Q THEN
					Sequence		:= 9999;
				END_IF;
            END_IF;
			            
        1000:    (* Menunggu Request *)
			Out_Rob_Placing := FALSE;
			CurrentJob		:= 'Waiting Request';
			Out_FB 			:= TRUE;
			Out_Req 		:= TRUE;
            IF Inp_Req AND Inp_FB AND (AccFlushing = 2 OR bBypassFGHS OR Data_Count_Real = 0) THEN
                Sequence := 1100;
            END_IF;
			
        1100:    (* Pallet Keluar *)
			CurrentJob		:= 'Pallet Out';
            Out_Motor_Rev	:= TRUE;
            IF (NOT Inp_SensorBack AND NOT Inp_SensorFront )AND NOT Inp_Req THEN
                DataTimer(IN := TRUE,PT := T#500ms);
                IF DataTimer.Q THEN
					TWatchDog(IN := FALSE);
					DataTimer(IN:=FALSE);
					Out_FB			:= FALSE;
					Out_Motor_Rev	:= FALSE;
                    Sequence		:= 1200;
                END_IF;
			ELSE
				TWatchDog(IN := TRUE, PT := T#15S);
				IF TWatchDog.Q THEN
					Sequence		:= 9999;
				END_IF;
            END_IF;
			
        1200:
			AccFlushing			:= 0;
			IF NOT Sts_Flushing THEN
			Data_Pallet_Total	:= Data_Pallet_Total + 1;
			END_IF
			Data_Count_Total	:= Data_Count_Total + Data_Count_Real;
			Sequence			:= 1300;
		   
        1300:
			CounterBarcode		:= 0;
            Data_Count_Real		:= 0;
			Data_Count_Place	:= 1;
			PalletID			:= '';
			PalletOut			:= TRUE;
            IF NOT Inp_Req THEN
                Sequence		:= 100;
            END_IF;
			
		9999:
			TWatchDog(IN := FALSE);
			DataTimer(IN:=FALSE);
			Out_PalletJammed	:= TRUE;
			Out_Motor_Rev 		:= FALSE;
			Out_Motor_Fwd 		:= FALSE;
			
        END_CASE;
ELSE
  	DataTimer(IN:=FALSE);
	TWatchDog(IN := FALSE);
	Out_Motor_Rev 		:= FALSE;
	Out_Motor_Fwd 		:= FALSE;
    Out_Rob_Placing 	:= FALSE;
    Out_Req 			:= FALSE;
	Out_FB 				:= FALSE;
	CurrentJob			:= 'Machine Stopped';
	IF Inp_GlobalReset THEN
        Sequence 		:= 0;
        Out_FB 			:= FALSE;
        Sts_Flushing 	:= FALSE;
    END_IF;
END_IF;

//Sequence Index
SeqIndex	:= Sequence;

IF Data_Count_Place = 0 THEN
    Data_Count_Place  := 1;
END_IF;

Data_Count_Place := Data_Count_Real+1;

// Calculate Max Cycle
o_MaxCycle :=i_Data*i_MaxStacking;

IF Inp_ResetData THEN
    Data_Count_Total	:= 0;
    Data_Pallet_Total 	:= 0;
    Data_Incomplete 	:= 0;
END_IF;

END_FUNCTION_BLOCK

// ---- POUs/Function_Block/Placing/PalletID_Name.TcPOU
FUNCTION_BLOCK PalletID_Name
VAR_INPUT
	CounterBox	: USINT;
	
	sYear		: STRING;
	sMonth		: STRING;
	sDate		: STRING;
	sHour		: STRING;
	sMinutes	: STRING;
	sSeconds	: STRING;
	PalletNumber: STRING(2);
	LineNumber	: STRING(2);
END_VAR
VAR_OUTPUT PERSISTENT
	PalletID	: STRING;
END_VAR
VAR
	Timer: TON;
END_VAR

VAR PERSISTENT
	PalletData: STRING;
	SeqIndex: INT;
END_VAR

PalletID:=PalletData;

CASE SeqIndex OF
	0:
		IF (CounterBox=1) THEN
			SeqIndex:=10;
		END_IF
	10:
		PalletData:=CONCAT(PalletNumber,CONCAT(sHour,CONCAT(sMinutes,CONCAT(sSeconds,CONCAT(sDate,CONCAT(sMonth,sYear))))));
		SeqIndex:=20;
	20:
		IF NOT (CounterBox=1) THEN
			SeqIndex:=0;
		END_IF
END_CASE

END_FUNCTION_BLOCK

// ---- POUs/Function_Block/General/MotorManagement.TcPOU
FUNCTION_BLOCK MotorManagement
VAR_IN_OUT
	Motor	: stMotor;
END_VAR

VAR_INPUT
	xIn_StatusDispatch	: BOOL;
	xIn_StatusError		: BOOL;
	xIn_StatusRunning	: BOOL;
	xIn_ResetError		: BOOL;
	xIn_AuxPower		: BOOL;
	UseReverse			: BOOL;
	TestMode			: BOOL;
	TriggerForward		: BOOL;
	TriggerReverse		: BOOL;
	
END_VAR
VAR_OUTPUT
	Error	: BOOL;
	ErrorID	: UINT;
END_VAR
VAR PERSISTENT
	StatusError			: BOOL;
	MotorCannotRunning	: BOOL;
	PowerOff			: BOOL;
	Timer				: TON;
	LocalSwitch_Off		: BOOL;
	SeqCal				: INT;
	tRunningHours		: LTIME;
	RunningTimer		: LTON;
	lrealRunningHours	: LREAL;
END_VAR
VAR // added by the converter: edge detectors and wires of the graphical bodies
    _w1 : BOOL;
END_VAR

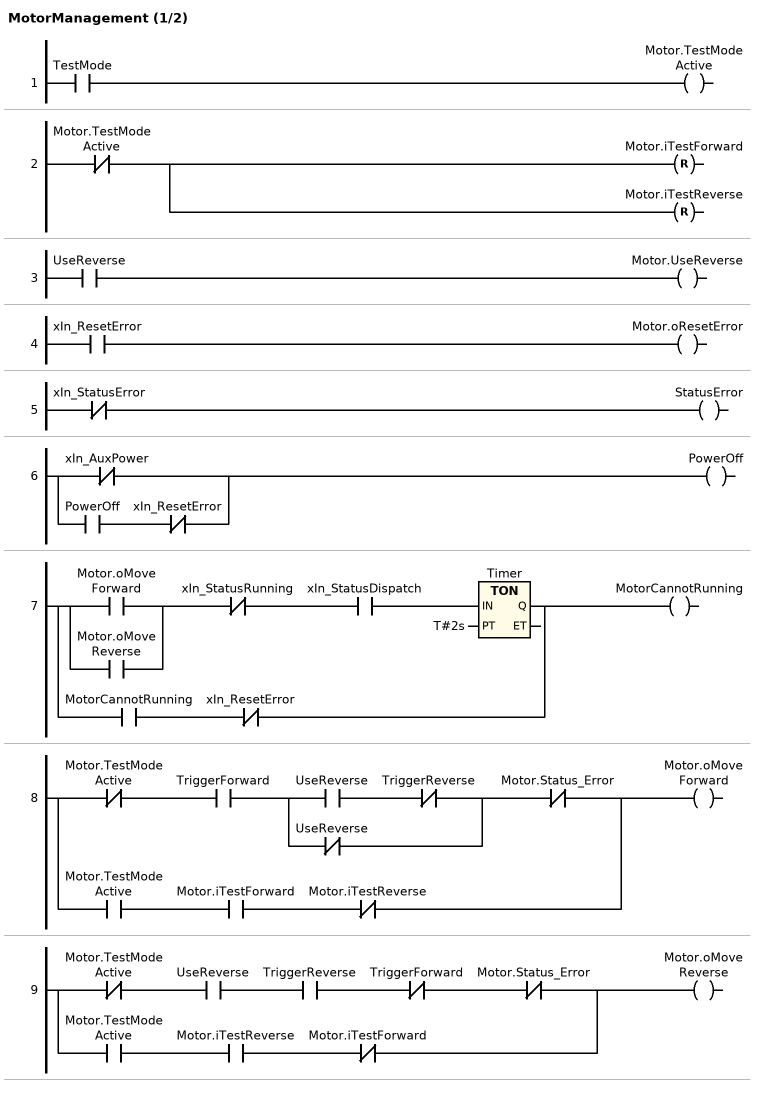
// NETWORK 1
Motor.TestModeActive := TestMode;

// NETWORK 2
_w1 := NOT Motor.TestModeActive;
Motor.iTestForward R= _w1;
Motor.iTestReverse R= _w1;

// NETWORK 3
Motor.UseReverse := UseReverse;

// NETWORK 4
Motor.oResetError := xIn_ResetError;

// NETWORK 5
StatusError := NOT xIn_StatusError;

// NETWORK 6
PowerOff := NOT xIn_AuxPower OR PowerOff AND NOT xIn_ResetError;

// NETWORK 7
Timer(IN := (Motor.oMoveForward OR Motor.oMoveReverse) AND NOT xIn_StatusRunning AND xIn_StatusDispatch, PT := T#2s); // TON
MotorCannotRunning := Timer.Q OR MotorCannotRunning AND NOT xIn_ResetError;

// NETWORK 8
Motor.oMoveForward := NOT Motor.TestModeActive AND TriggerForward AND (UseReverse AND NOT TriggerReverse OR NOT UseReverse) AND NOT Motor.Status_Error OR Motor.TestModeActive AND Motor.iTestForward AND NOT Motor.iTestReverse;

// NETWORK 9
Motor.oMoveReverse := NOT Motor.TestModeActive AND UseReverse AND TriggerReverse AND NOT TriggerForward AND NOT Motor.Status_Error OR Motor.TestModeActive AND Motor.iTestReverse AND NOT Motor.iTestForward;

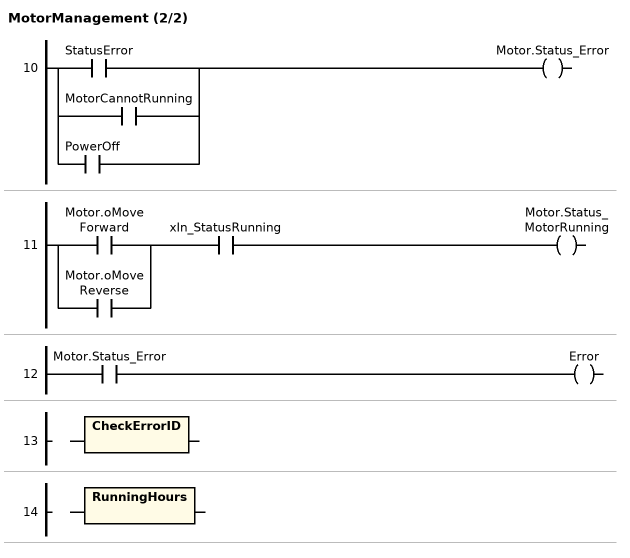
// NETWORK 10
Motor.Status_Error := StatusError OR MotorCannotRunning OR PowerOff;

// NETWORK 11
Motor.Status_MotorRunning := (Motor.oMoveForward OR Motor.oMoveReverse) AND xIn_StatusRunning;

// NETWORK 12
Error := Motor.Status_Error;

// NETWORK 13
CheckErrorID();

// NETWORK 14
RunningHours();

ACTION CheckErrorID:
IF Error THEN
	IF StatusError THEN
		ErrorID:=1;
	ELSIF PowerOff THEN
			ErrorID:=2;
		ELSIF LocalSwitch_Off THEN
				ErrorID:=3;
			ELSIF MotorCannotRunning THEN
					ErrorID:=10;
				ELSE
					ErrorID:=90;
			END_IF
ELSE
	ErrorID:=0;
END_IF

Motor.ErrorID:=ErrorID;
END_ACTION

ACTION RunningHours:
CASE SeqCal OF
	0:
		Motor.RunningTime	:= tRunningHours;
		IF Motor.Status_MotorRunning THEN
			SeqCal	:= 1;
		END_IF
		
	1:
		RunningTimer(IN:=TRUE,PT:=LTIME#1H);
		Motor.RunningTime	:= tRunningHours + RunningTimer.ET;
		IF RunningTimer.Q OR NOT Motor.Status_MotorRunning THEN
			RunningTimer(IN:=FALSE);
			SeqCal	:= 2;
		END_IF
		
	2:
		tRunningHours	:= Motor.RunningTime;
		SeqCal			:= 0;
END_CASE

Motor.RunningHours	:= LTIME_TO_LREAL(Motor.RunningTime) / LTIME_TO_LREAL(LTIME#1H);
END_ACTION

END_FUNCTION_BLOCK

// ---- POUs/Function/ConvertMilliSecTimeData.TcPOU
FUNCTION ConvertMilliSecTimeData : TIME
VAR_INPUT
	DataInput	: UINT;
END_VAR
VAR
END_VAR

ConvertMilliSecTimeData:=LINT_TO_TIME(UINT_TO_LINT(DataInput));

END_FUNCTION

// ---- POUs/S02_Placing/EM03_Placing2.TcPOU
PROGRAM EM03_Placing2
VAR
	
	//Backbone
	FB_StateMachine_Placing2		: FB_StateManager;
	bFl_RunningMachinePlacing2		: BOOL;
	bFl_SeqReset					: BOOL;
	bFl_Manual						: BOOL;
	CheckStatusPlacing2				: checkstatus;
	AlarmEventHistory				: ARRAY[1..20] OF Alarm_Event_History;
	Placing2_Management				: FB_Placing;
	bFl_Flushing					: BOOL;
	PalletID_Placing2				: PalletID_Name;
	Placing2_ID						: STRING;
	bFl_PalletJammed				: BOOL;
	
	//Motor
	Motor_PalletPlacing2			: MotorManagement;
	bFl_MotorPlacing2				: BOOL;
	Motor_Placing2_Error			: BOOL;
	Motor_Placing2_ErrorID			: UINT;
	bFl_MotorPlacing2_Fwd			: BOOL;
	bFl_MotorPlacing2_Rev			: BOOL;
	bFL_Safety						: BOOL;
	AlarmEventActive				: ARRAY[1..20] OF Alarm_Event_Active;
	CheckAcc						: TON;
END_VAR
VAR // added by the converter: edge detectors and wires of the graphical bodies
    _w1 : BOOL;
END_VAR

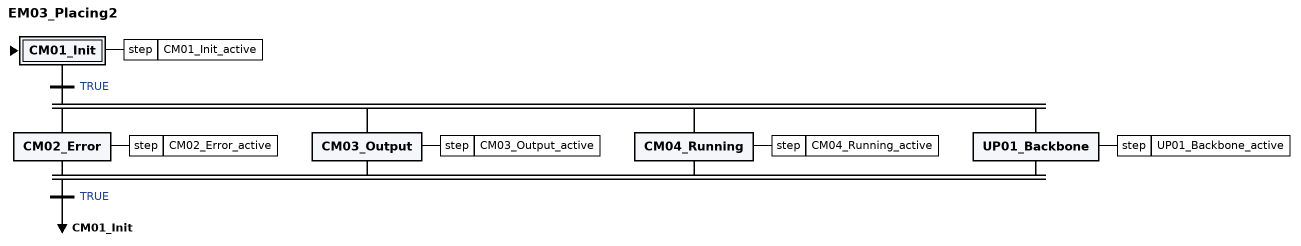
INITIAL_STEP CM01_Init:
    CM01_Init_active(N);  // step action
END_STEP
TRANSITION FROM CM01_Init TO (CM02_Error, CM03_Output, CM04_Running, UP01_Backbone)
    := TRUE;
END_TRANSITION
STEP CM02_Error:
    CM02_Error_active(N);  // step action
END_STEP
STEP CM03_Output:
    CM03_Output_active(N);  // step action
END_STEP
STEP CM04_Running:
    CM04_Running_active(N);  // step action
END_STEP
STEP UP01_Backbone:
    UP01_Backbone_active(N);  // step action
END_STEP
TRANSITION FROM (CM02_Error, CM03_Output, CM04_Running, UP01_Backbone) TO CM01_Init
    := TRUE;
END_TRANSITION

ACTION CM01_Init_active:
Data_GVL.bFL_StartPlacing2			:= Status_GVL.bFl_RunButton_Robotic OR HMI_GVL.bStartButtonPlacing2;
Data_GVL.bFL_StopPlacing2			:= NOT Status_GVL.bFl_StopButton_Robotic OR HMI_GVL.bStopButtonPlacing2;
Data_GVL.bFL_ResetPlacing2			:= Status_GVL.bFl_ResetButton_Robotic OR HMI_GVL.bResetButtonPlacing2;
Data_GVL.bFL_AckPlacing2			:= Status_GVL.bFl_Acknowledge_Robotic OR HMI_GVL.bAcknowledgeButtonPlacing2;
Data_GVL.bFL_AutoManuaModePlacing2 	:= Status_GVL.bFl_Manual_Robotic OR HMI_GVL.bTestModeEnablePlacing2;
bFl_RunningMachinePlacing2			:= Data_GVL.stStateMachinePlacing2.Running;
bFl_Manual							:= Data_GVL.stStateMachinePlacing2.ManualMode;
bFl_SeqReset						:= NOT Status_GVL.bFl_EStop_Robotic;
bFL_Safety							:= Status_GVL.bFl_EStop_Robotic AND Status_GVL.bSafety_DoorRobotic;


(*=================Convert Timer============================*)
Data_GVL.Tmr_Placing2	:= ConvertMilliSecTimeData(HMI_GVL.Tmr_Placing2);

(*=================Data OEE============================*)
Data_GVL.dt_Production[2].Data1			:= HMI_GVL.arCountTotal[2];
Data_GVL.dt_Production[2].Data2			:= HMI_GVL.arPalletTotal[2];
Data_GVL.dt_Production[2].Data3			:= HMI_GVL.arPalletIncomplete[2];
Data_GVL.dt_Production[2].ProductCode	:= Status_GVL.RecipeLine[2].ProductName;
END_ACTION

ACTION CM02_Error_active:
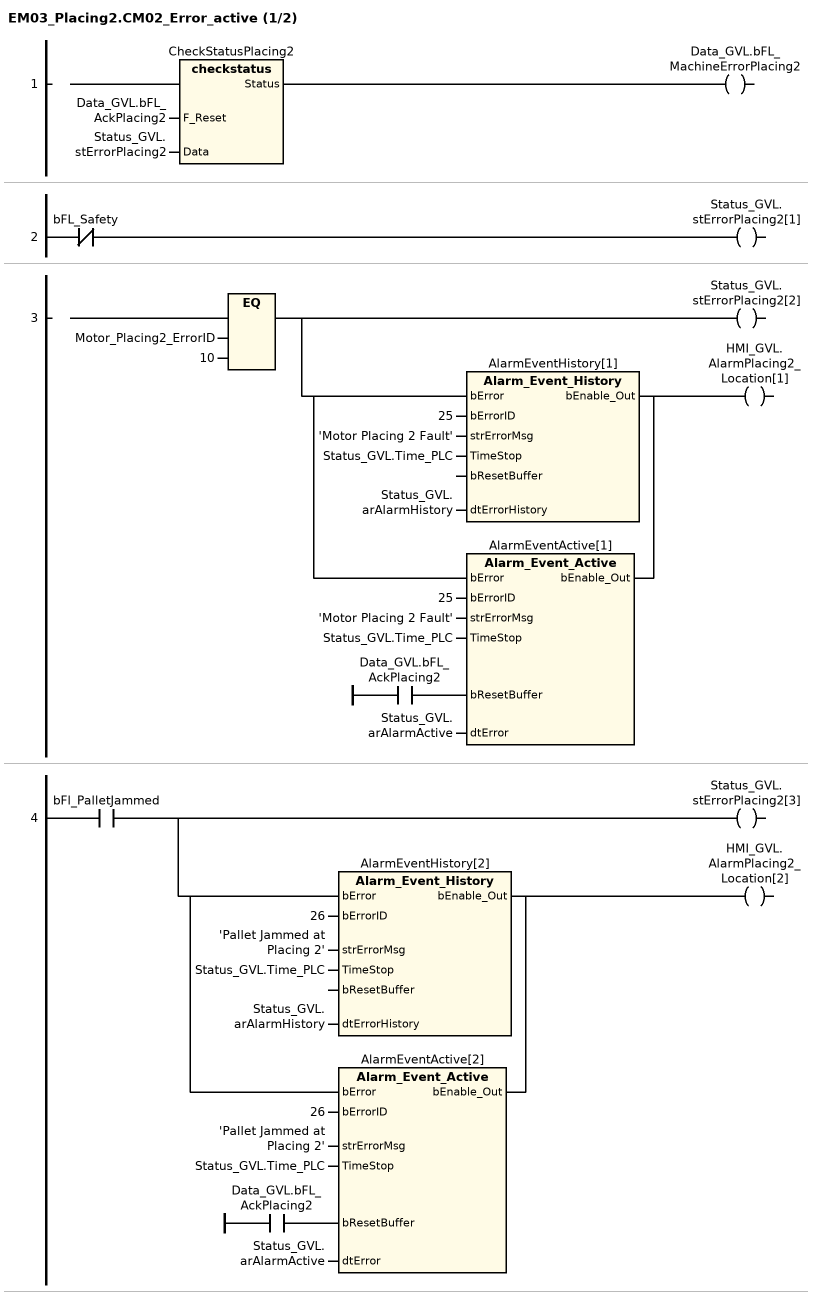
// NETWORK 1
CheckStatusPlacing2(F_Reset := Data_GVL.bFL_AckPlacing2, Data := Status_GVL.stErrorPlacing2); // checkstatus
Data_GVL.bFL_MachineErrorPlacing2 := CheckStatusPlacing2.Status;

// NETWORK 2
Status_GVL.stErrorPlacing2[1] := NOT bFL_Safety;

// NETWORK 3
_w1 := Motor_Placing2_ErrorID = 10;
Status_GVL.stErrorPlacing2[2] := _w1;
AlarmEventHistory[1](
    bError := _w1,
    bErrorID := 25,
    strErrorMsg := 'Motor Placing 2 Fault',
    TimeStop := Status_GVL.Time_PLC,
    dtErrorHistory := Status_GVL.arAlarmHistory); // Alarm_Event_History
AlarmEventActive[1](
    bError := _w1,
    bErrorID := 25,
    strErrorMsg := 'Motor Placing 2 Fault',
    TimeStop := Status_GVL.Time_PLC,
    bResetBuffer := Data_GVL.bFL_AckPlacing2,
    dtError := Status_GVL.arAlarmActive); // Alarm_Event_Active
HMI_GVL.AlarmPlacing2_Location[1] := AlarmEventHistory[1].bEnable_Out OR AlarmEventActive[1].bEnable_Out;

// NETWORK 4
Status_GVL.stErrorPlacing2[3] := bFl_PalletJammed;
AlarmEventHistory[2](
    bError := bFl_PalletJammed,
    bErrorID := 26,
    strErrorMsg := 'Pallet Jammed at Placing 2',
    TimeStop := Status_GVL.Time_PLC,
    dtErrorHistory := Status_GVL.arAlarmHistory); // Alarm_Event_History
AlarmEventActive[2](
    bError := bFl_PalletJammed,
    bErrorID := 26,
    strErrorMsg := 'Pallet Jammed at Placing 2',
    TimeStop := Status_GVL.Time_PLC,
    bResetBuffer := Data_GVL.bFL_AckPlacing2,
    dtError := Status_GVL.arAlarmActive); // Alarm_Event_Active
HMI_GVL.AlarmPlacing2_Location[2] := AlarmEventHistory[2].bEnable_Out OR AlarmEventActive[2].bEnable_Out;

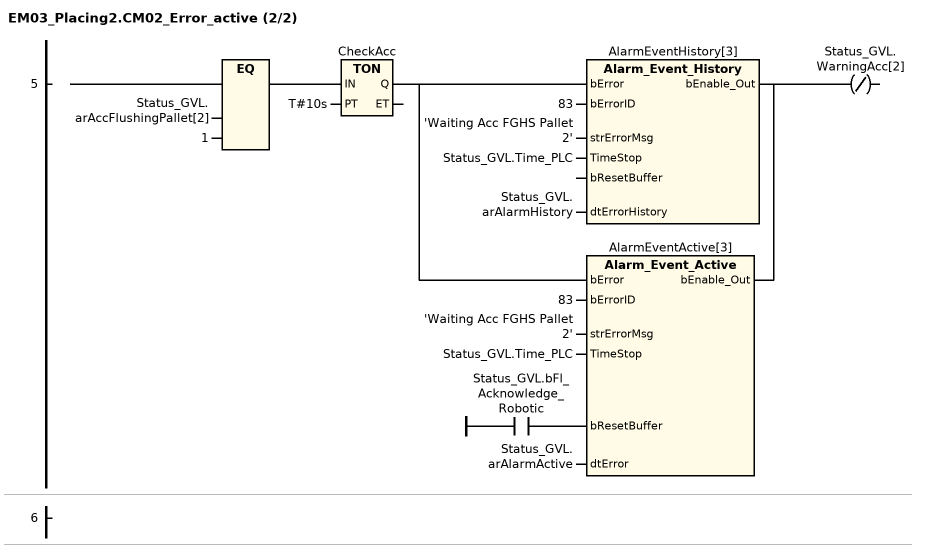
// NETWORK 5
CheckAcc(IN := Status_GVL.arAccFlushingPallet[2] = 1, PT := T#10s); // TON
AlarmEventHistory[3](
    bError := CheckAcc.Q,
    bErrorID := 83,
    strErrorMsg := 'Waiting Acc FGHS Pallet 2',
    TimeStop := Status_GVL.Time_PLC,
    dtErrorHistory := Status_GVL.arAlarmHistory); // Alarm_Event_History
AlarmEventActive[3](
    bError := CheckAcc.Q,
    bErrorID := 83,
    strErrorMsg := 'Waiting Acc FGHS Pallet 2',
    TimeStop := Status_GVL.Time_PLC,
    bResetBuffer := Status_GVL.bFl_Acknowledge_Robotic,
    dtError := Status_GVL.arAlarmActive); // Alarm_Event_Active
Status_GVL.WarningAcc[2] := NOT (AlarmEventHistory[3].bEnable_Out OR AlarmEventActive[3].bEnable_Out);

// NETWORK 6
END_ACTION

ACTION CM03_Output_active:
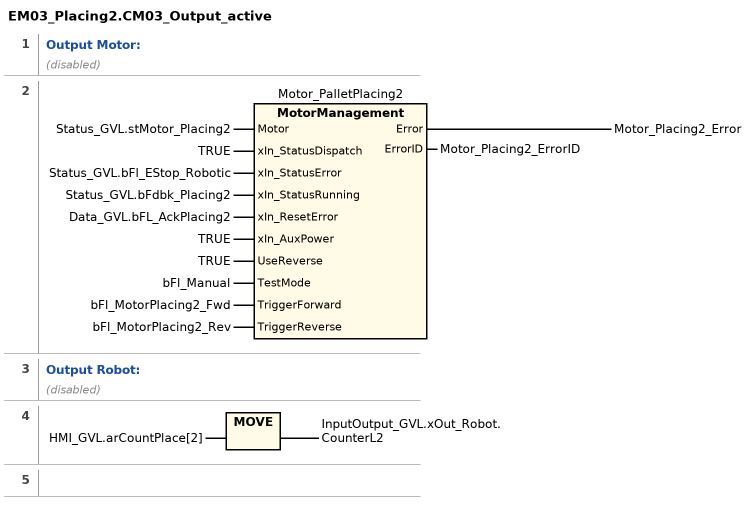
// NETWORK 1 (disabled)
// label: Output Motor

// NETWORK 2
Motor_PalletPlacing2(
    Motor := Status_GVL.stMotor_Placing2,
    xIn_StatusDispatch := TRUE,
    xIn_StatusError := Status_GVL.bFl_EStop_Robotic,
    xIn_StatusRunning := Status_GVL.bFdbk_Placing2,
    xIn_ResetError := Data_GVL.bFL_AckPlacing2,
    xIn_AuxPower := TRUE,
    UseReverse := TRUE,
    TestMode := bFl_Manual,
    TriggerForward := bFl_MotorPlacing2_Fwd,
    TriggerReverse := bFl_MotorPlacing2_Rev,
    ErrorID => Motor_Placing2_ErrorID); // MotorManagement
Motor_Placing2_Error := Motor_PalletPlacing2.Error;

// NETWORK 3 (disabled)
// label: Output Robot

// NETWORK 4
InputOutput_GVL.xOut_Robot.CounterL2 := HMI_GVL.arCountPlace[2];

// NETWORK 5
END_ACTION

ACTION CM04_Running_active:
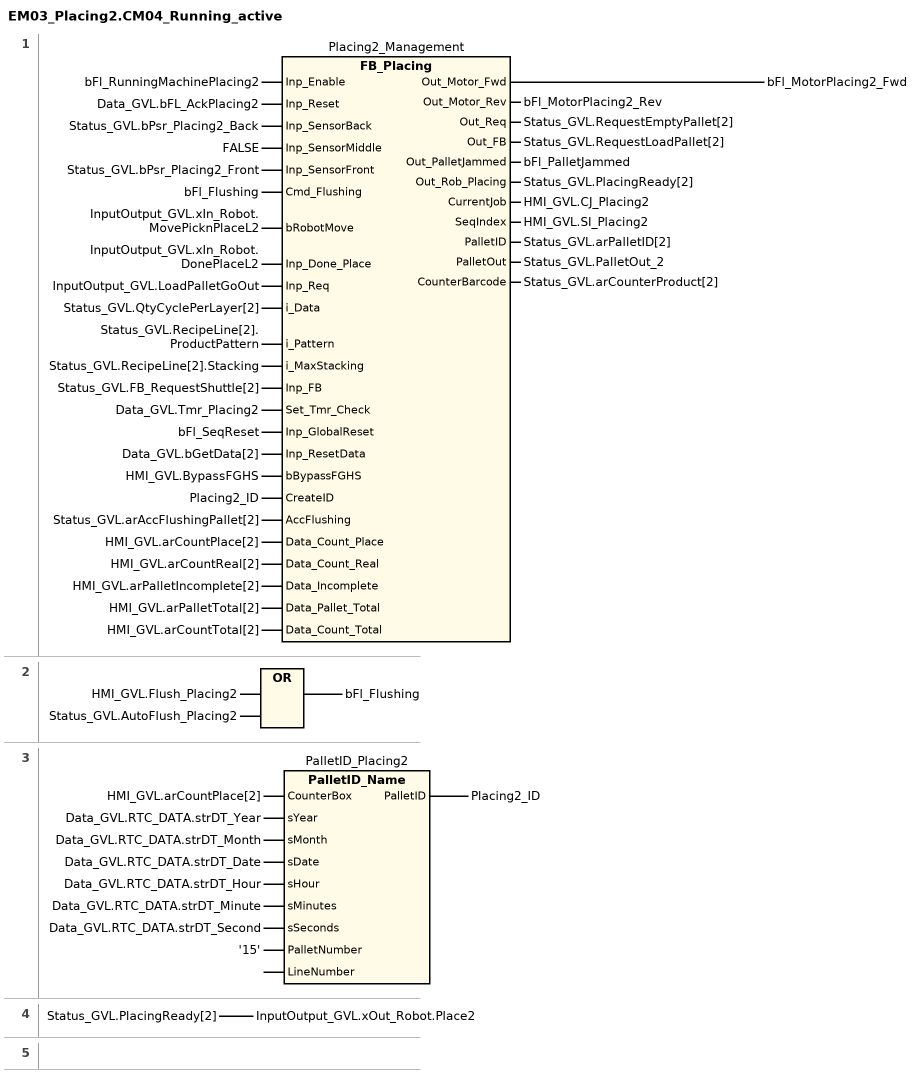
// NETWORK 1
Placing2_Management(
    Inp_Enable := bFl_RunningMachinePlacing2,
    Inp_Reset := Data_GVL.bFL_AckPlacing2,
    Inp_SensorBack := Status_GVL.bPsr_Placing2_Back,
    Inp_SensorMiddle := FALSE,
    Inp_SensorFront := Status_GVL.bPsr_Placing2_Front,
    Cmd_Flushing := bFl_Flushing,
    bRobotMove := InputOutput_GVL.xIn_Robot.MovePicknPlaceL2,
    Inp_Done_Place := InputOutput_GVL.xIn_Robot.DonePlaceL2,
    Inp_Req := InputOutput_GVL.LoadPalletGoOut,
    i_Data := Status_GVL.QtyCyclePerLayer[2],
    i_Pattern := Status_GVL.RecipeLine[2].ProductPattern,
    i_MaxStacking := Status_GVL.RecipeLine[2].Stacking,
    Inp_FB := Status_GVL.FB_RequestShuttle[2],
    Set_Tmr_Check := Data_GVL.Tmr_Placing2,
    Inp_GlobalReset := bFl_SeqReset,
    Inp_ResetData := Data_GVL.bGetData[2],
    bBypassFGHS := HMI_GVL.BypassFGHS,
    CreateID := Placing2_ID,
    AccFlushing := Status_GVL.arAccFlushingPallet[2],
    Data_Count_Place := HMI_GVL.arCountPlace[2],
    Data_Count_Real := HMI_GVL.arCountReal[2],
    Data_Incomplete := HMI_GVL.arPalletIncomplete[2],
    Data_Pallet_Total := HMI_GVL.arPalletTotal[2],
    Data_Count_Total := HMI_GVL.arCountTotal[2],
    Out_Motor_Rev => bFl_MotorPlacing2_Rev,
    Out_Req => Status_GVL.RequestEmptyPallet[2],
    Out_FB => Status_GVL.RequestLoadPallet[2],
    Out_PalletJammed => bFl_PalletJammed,
    Out_Rob_Placing => Status_GVL.PlacingReady[2],
    CurrentJob => HMI_GVL.CJ_Placing2,
    SeqIndex => HMI_GVL.SI_Placing2,
    PalletID => Status_GVL.arPalletID[2],
    PalletOut => Status_GVL.PalletOut_2,
    CounterBarcode => Status_GVL.arCounterProduct[2]); // FB_Placing
bFl_MotorPlacing2_Fwd := Placing2_Management.Out_Motor_Fwd;

// NETWORK 2
bFl_Flushing := HMI_GVL.Flush_Placing2 OR Status_GVL.AutoFlush_Placing2;

// NETWORK 3
PalletID_Placing2(
    CounterBox := HMI_GVL.arCountPlace[2],
    sYear := Data_GVL.RTC_DATA.strDT_Year,
    sMonth := Data_GVL.RTC_DATA.strDT_Month,
    sDate := Data_GVL.RTC_DATA.strDT_Date,
    sHour := Data_GVL.RTC_DATA.strDT_Hour,
    sMinutes := Data_GVL.RTC_DATA.strDT_Minute,
    sSeconds := Data_GVL.RTC_DATA.strDT_Second,
    PalletNumber := '15'); // PalletID_Name
Placing2_ID := PalletID_Placing2.PalletID;

// NETWORK 4
InputOutput_GVL.xOut_Robot.Place2 := Status_GVL.PlacingReady[2];

// NETWORK 5
END_ACTION

ACTION UP01_Backbone_active:
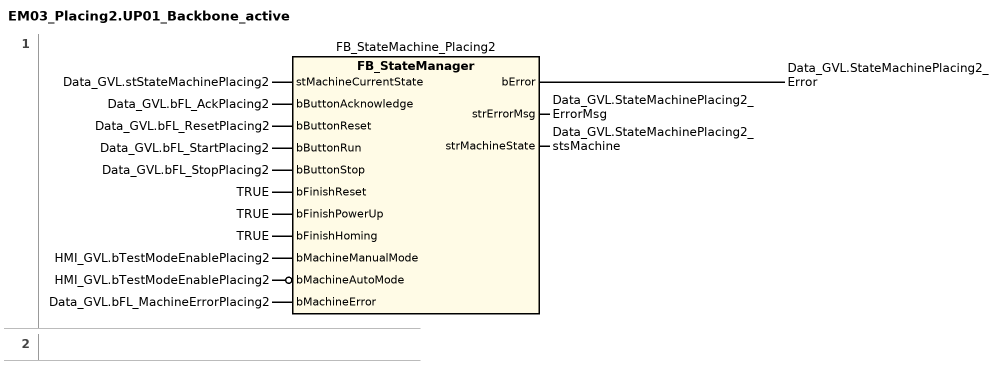
// NETWORK 1
FB_StateMachine_Placing2(
    stMachineCurrentState := Data_GVL.stStateMachinePlacing2,
    bButtonAcknowledge := Data_GVL.bFL_AckPlacing2,
    bButtonReset := Data_GVL.bFL_ResetPlacing2,
    bButtonRun := Data_GVL.bFL_StartPlacing2,
    bButtonStop := Data_GVL.bFL_StopPlacing2,
    bFinishReset := TRUE,
    bFinishPowerUp := TRUE,
    bFinishHoming := TRUE,
    bMachineManualMode := HMI_GVL.bTestModeEnablePlacing2,
    bMachineAutoMode := NOT HMI_GVL.bTestModeEnablePlacing2,
    bMachineError := Data_GVL.bFL_MachineErrorPlacing2,
    strErrorMsg => Data_GVL.StateMachinePlacing2_ErrorMsg,
    strMachineState => Data_GVL.StateMachinePlacing2_stsMachine); // FB_StateManager
Data_GVL.StateMachinePlacing2_Error := FB_StateMachine_Placing2.bError;

// NETWORK 2
END_ACTION

END_PROGRAM

// ---- POUs/Function_Block/Placing/FB_Placing.TcPOU
FUNCTION_BLOCK FB_Placing
VAR_INPUT
	Inp_Enable				: BOOL;
	Inp_Reset				: BOOL;
	Inp_SensorBack			: BOOL;
	Inp_SensorMiddle		: BOOL;
	Inp_SensorFront			: BOOL;
	Cmd_Flushing			: BOOL;
	bRobotMove				: BOOL;
	Inp_Done_Place			: BOOL;
	Inp_Req					: BOOL;
	i_Data					: UINT;
	i_Pattern				: UINT;
	i_MaxStacking			: UINT;
	Inp_FB					: BOOL;
	Set_Tmr_Check			: TIME;
	Inp_GlobalReset			: BOOL;
	Inp_ResetData			: BOOL;
	bBypassFGHS				: BOOL;
	CreateID				: STRING;
	
END_VAR
VAR_OUTPUT
	Out_Motor_Fwd			: BOOL;
	Out_Motor_Rev			: BOOL;
	Out_Req					: BOOL;
	Out_FB					: BOOL;
	Out_PalletJammed		: BOOL;
	Out_Rob_Placing			: BOOL;
	CurrentJob				: STRING;
	SeqIndex				: INT;
	PalletOut				: BOOL;
END_VAR
VAR_OUTPUT PERSISTENT
	PalletID				: STRING;
	CounterBarcode			: BYTE;
END_VAR

VAR
	Sts_Flushing			: BOOL;
	o_MaxCycle				: UINT;
	DataTimer				: TON;
	TWatchDog				: TON;
	Sequence				: INT;
END_VAR

VAR_IN_OUT
	AccFlushing				: BYTE;
	Data_Count_Place		: USINT;
	Data_Count_Real			: USINT;
	Data_Incomplete			: UINT;
	Data_Pallet_Total		: UINT;
	Data_Count_Total		: UINT;
END_VAR

IF Inp_Reset AND Out_PalletJammed THEN
	Out_PalletJammed	:= FALSE;
	Sequence 			:= 0;
END_IF

IF Inp_Enable THEN
	
	IF Cmd_Flushing THEN
		Sts_Flushing:=TRUE;
	END_IF;
	
    CASE Sequence OF
        0:	(* Check Motor *)
			 Out_Motor_Fwd := TRUE;
			 DataTimer(IN:=TRUE, PT:=T#4S);
			 IF DataTimer.Q THEN
				 DataTimer(IN:=FALSE);
				 Out_Motor_Fwd	:= FALSE;
				 Sequence		:= 10;
			 END_IF

		10:  (* Check Sensor *)
			CurrentJob		:= 'Check Sensor';
			IF (Inp_SensorFront OR Inp_SensorMiddle OR Inp_SensorBack) AND AccFlushing = 2 THEN
				Sequence := 600;
			ELSIF (Inp_SensorFront OR Inp_SensorMiddle OR Inp_SensorBack) AND ((Data_Count_Place > o_MaxCycle AND o_MaxCycle <> 0)  OR Sts_Flushing) THEN
                Sequence := 500;
            ELSIF Inp_SensorFront THEN
                Sequence := 300;
            ELSIF NOT Inp_SensorFront AND (Inp_SensorMiddle OR Inp_SensorBack)  THEN
                Sequence := 200;
            ELSE
                Sequence := 100;
            END_IF;
			
			
        100:    (* Request *)
			CurrentJob		:= 'Request Pallet';
			Sts_Flushing	:= FALSE;
            Out_Req			:= TRUE;
			Out_FB			:= FALSE;
            IF Inp_FB THEN
				DataTimer(IN:=FALSE);
                Sequence := 200;
            END_IF;       
			
        200:    (* Pallet Masuk *)
			CurrentJob	:= 'Pallet In';
			PalletOut	:= FALSE;
			IF NOT Inp_SensorFront AND NOT Inp_SensorMiddle AND NOT Inp_SensorBack THEN
            	Out_Req := TRUE;
			END_IF
            Out_Motor_Fwd := TRUE;
            IF Inp_SensorFront AND (Inp_SensorBack OR Inp_SensorMiddle)  THEN
				DataTimer(IN := TRUE,PT := Set_Tmr_Check);
                IF DataTimer.Q THEN
					TWatchDog(IN := FALSE);
                    DataTimer(IN:=FALSE);
					Out_PalletJammed	:= FALSE;
					Out_Motor_Fwd		:= FALSE;
           			Out_Req				:= FALSE;
                    Sequence			:= 300;
                END_IF;    
			ELSE
				TWatchDog(IN := TRUE, PT := T#30S);
				IF TWatchDog.Q THEN
					Sequence	:= 9999;
				END_IF;
            END_IF;
			
        300:
			CurrentJob	:= 'Check Cycle';
			IF o_MaxCycle <> 0 THEN
				IF o_MaxCycle >= Data_Count_Place  THEN
					Sequence := 400;
				ELSE
					DataTimer(IN := TRUE,PT := T#2S);
					IF DataTimer.Q THEN
						DataTimer(IN:=FALSE);
						Sequence := 500;
					END_IF;
				END_IF;
			END_IF
			
        400:
			CurrentJob		:= 'Place Ready';
			AccFlushing		:= 0;
            Out_Rob_Placing := TRUE;
			PalletID		:= CreateID;
            IF Inp_Done_Place THEN
                    Data_Count_Real		:= Data_Count_Real + 1;
                    Data_Count_Place	:= Data_Count_Place + 1;
                    Sequence 			:= 450;
            ELSIF (Cmd_Flushing OR Sts_Flushing) AND NOT bRobotMove THEN
                Data_Incomplete			:= Data_Incomplete + 1;
                Sts_Flushing			:= TRUE;
                Sequence 				:= 500;				
            END_IF;
			
        450:
            Out_Rob_Placing := FALSE;
            IF NOT Inp_Done_Place THEN
                Sequence := 460;
            END_IF;	
			
		460:
			IF PalletID <> '' THEN
				CounterBarcode	:= Data_Count_Real;
				Sequence 		:= 300;
			END_IF
			
		500:
			
			CurrentJob		:= 'Create Pallet ID';
			DataTimer(IN := TRUE,PT := T#500MS);
			IF DataTimer.Q THEN
				DataTimer(IN := FALSE);
				Sequence		:= 550;
			END_IF
						
		550:
			AccFlushing		:= 1;
			Sequence		:= 600;
			
		600:
			Out_Rob_Placing := FALSE;
			Out_FB 			:= FALSE;
			Out_Req 		:= FALSE;
			CurrentJob		:= 'Waiting Acc Flushing';
			IF (PalletID <> '' AND AccFlushing = 2) OR bBypassFGHS OR Data_Count_Real = 0 THEN
                Sequence := 1000;
            END_IF;
		
            
        1000:    (* Menunggu Request *)
			Out_Rob_Placing := FALSE;
			CurrentJob		:= 'Waiting Request';
			Out_FB 			:= TRUE;
			Out_Req 		:= TRUE;
            IF Inp_Req AND Inp_FB AND (AccFlushing = 2 OR bBypassFGHS OR Data_Count_Real = 0)  THEN
                Sequence := 1100;
            END_IF;
			
        1100:    (* Pallet Keluar *)
			CurrentJob		:= 'Pallet Out';
            Out_Motor_Rev	:= TRUE;
            IF (NOT Inp_SensorBack AND NOT Inp_SensorFront )AND NOT Inp_Req THEN
                DataTimer(IN := TRUE,PT := T#500ms);
                IF DataTimer.Q THEN
					TWatchDog(IN := FALSE);
					DataTimer(IN:=FALSE);
					Out_FB			:= FALSE;
					Out_Motor_Rev	:= FALSE;
                    Sequence		:= 1200;
                END_IF;
			ELSE
				TWatchDog(IN := TRUE, PT := T#15S);
				IF TWatchDog.Q THEN
					Sequence		:= 9999;
				END_IF;
            END_IF;
			
        1200:
			AccFlushing			:= 0;
			IF NOT Sts_Flushing THEN
			Data_Pallet_Total	:= Data_Pallet_Total + 1;
			END_IF
			Data_Count_Total	:= Data_Count_Total + Data_Count_Real;
			Sequence			:= 1300;
		   
        1300:
			CounterBarcode		:= 0;
            Data_Count_Real		:= 0;
			Data_Count_Place	:= 1;
			PalletID			:= '';
			PalletOut			:= TRUE;
            IF NOT Inp_Req THEN
                Sequence		:= 100;
            END_IF;
			
		9999:
			TWatchDog(IN := FALSE);
			DataTimer(IN:=FALSE);
			Out_PalletJammed	:= TRUE;
			Out_Motor_Rev 		:= FALSE;
			Out_Motor_Fwd 		:= FALSE;
			
        END_CASE;
ELSE
  	DataTimer(IN:=FALSE);
	TWatchDog(IN := FALSE);
	Out_Motor_Rev 		:= FALSE;
	Out_Motor_Fwd 		:= FALSE;
    Out_Rob_Placing 	:= FALSE;
    Out_Req 			:= FALSE;
	Out_FB 				:= FALSE;
	CurrentJob			:= 'Machine Stopped';
	IF Inp_GlobalReset THEN
        Sequence 		:= 0;
        Out_FB 			:= FALSE;
        Sts_Flushing 	:= FALSE;
    END_IF;
END_IF;

//Sequence Index
SeqIndex	:= Sequence;

IF Data_Count_Place = 0 THEN
    Data_Count_Place  := 1;
END_IF;

Data_Count_Place := Data_Count_Real+1;

// Calculate Max Cycle
o_MaxCycle :=i_Data*i_MaxStacking;

IF Inp_ResetData THEN
    Data_Count_Total	:= 0;
    Data_Pallet_Total 	:= 0;
    Data_Incomplete 	:= 0;
END_IF;

END_FUNCTION_BLOCK

// ---- POUs/S02_Placing/EM04_Placing3.TcPOU
PROGRAM EM04_Placing3
VAR
	
	//Backbone
	FB_StateMachine_Placing3		: FB_StateManager;
	bFl_RunningMachinePlacing3		: BOOL;
	bFl_SeqReset					: BOOL;
	bFl_Manual						: BOOL;
	CheckStatusPlacing3				: checkstatus;
	AlarmEventHistory				: ARRAY[1..20] OF Alarm_Event_History;
	Placing3_Management				: FB_Placing;
	bFl_Flushing					: BOOL;
	PalletID_Placing3				: PalletID_Name;
	Placing3_ID						: STRING;
	bFl_PalletJammed				: BOOL;
	
	//Motor
	Motor_PalletPlacing3			: MotorManagement;
	bFl_MotorPlacing3				: BOOL;
	Motor_Placing3_Error			: BOOL;
	Motor_Placing3_ErrorID			: UINT;
	bFl_MotorPlacing3_Fwd			: BOOL;
	bFl_MotorPlacing3_Rev			: BOOL;
	bFL_Safety						: BOOL;
	AlarmEventActive				: ARRAY[1..20] OF Alarm_Event_Active;
	CheckAcc						: TON;
END_VAR
VAR // added by the converter: edge detectors and wires of the graphical bodies
    _w1 : BOOL;
END_VAR

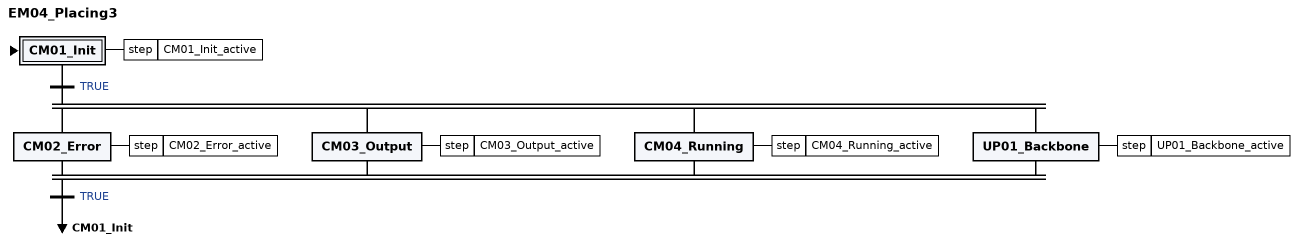
INITIAL_STEP CM01_Init:
    CM01_Init_active(N);  // step action
END_STEP
TRANSITION FROM CM01_Init TO (CM02_Error, CM03_Output, CM04_Running, UP01_Backbone)
    := TRUE;
END_TRANSITION
STEP CM02_Error:
    CM02_Error_active(N);  // step action
END_STEP
STEP CM03_Output:
    CM03_Output_active(N);  // step action
END_STEP
STEP CM04_Running:
    CM04_Running_active(N);  // step action
END_STEP
STEP UP01_Backbone:
    UP01_Backbone_active(N);  // step action
END_STEP
TRANSITION FROM (CM02_Error, CM03_Output, CM04_Running, UP01_Backbone) TO CM01_Init
    := TRUE;
END_TRANSITION

ACTION CM01_Init_active:
Data_GVL.bFL_StartPlacing3			:= Status_GVL.bFl_RunButton_Robotic OR HMI_GVL.bStartButtonPlacing3;
Data_GVL.bFL_StopPlacing3			:= NOT Status_GVL.bFl_StopButton_Robotic OR HMI_GVL.bStopButtonPlacing3;
Data_GVL.bFL_ResetPlacing3			:= Status_GVL.bFl_ResetButton_Robotic OR HMI_GVL.bResetButtonPlacing3;
Data_GVL.bFL_AckPlacing3			:= Status_GVL.bFl_Acknowledge_Robotic OR HMI_GVL.bAcknowledgeButtonPlacing3;
Data_GVL.bFL_AutoManuaModePlacing3 	:= Status_GVL.bFl_Manual_Robotic OR HMI_GVL.bTestModeEnablePlacing3;
bFl_RunningMachinePlacing3			:= Data_GVL.stStateMachinePlacing3.Running;
bFl_Manual							:= Data_GVL.stStateMachinePlacing3.ManualMode;
bFl_SeqReset						:= NOT Status_GVL.bFl_EStop_Robotic;
bFL_Safety							:= Status_GVL.bFl_EStop_Robotic AND Status_GVL.bSafety_DoorRobotic;


(*=================Convert Timer============================*)
Data_GVL.Tmr_Placing3	:= ConvertMilliSecTimeData(HMI_GVL.Tmr_Placing3);


(*=================Data OEE============================*)
Data_GVL.dt_Production[3].Data1			:= HMI_GVL.arCountTotal[3];
Data_GVL.dt_Production[3].Data2			:= HMI_GVL.arPalletTotal[3];
Data_GVL.dt_Production[3].Data3			:= HMI_GVL.arPalletIncomplete[3];
Data_GVL.dt_Production[3].ProductCode	:= Status_GVL.RecipeLine[3].ProductName;
END_ACTION

ACTION CM02_Error_active:
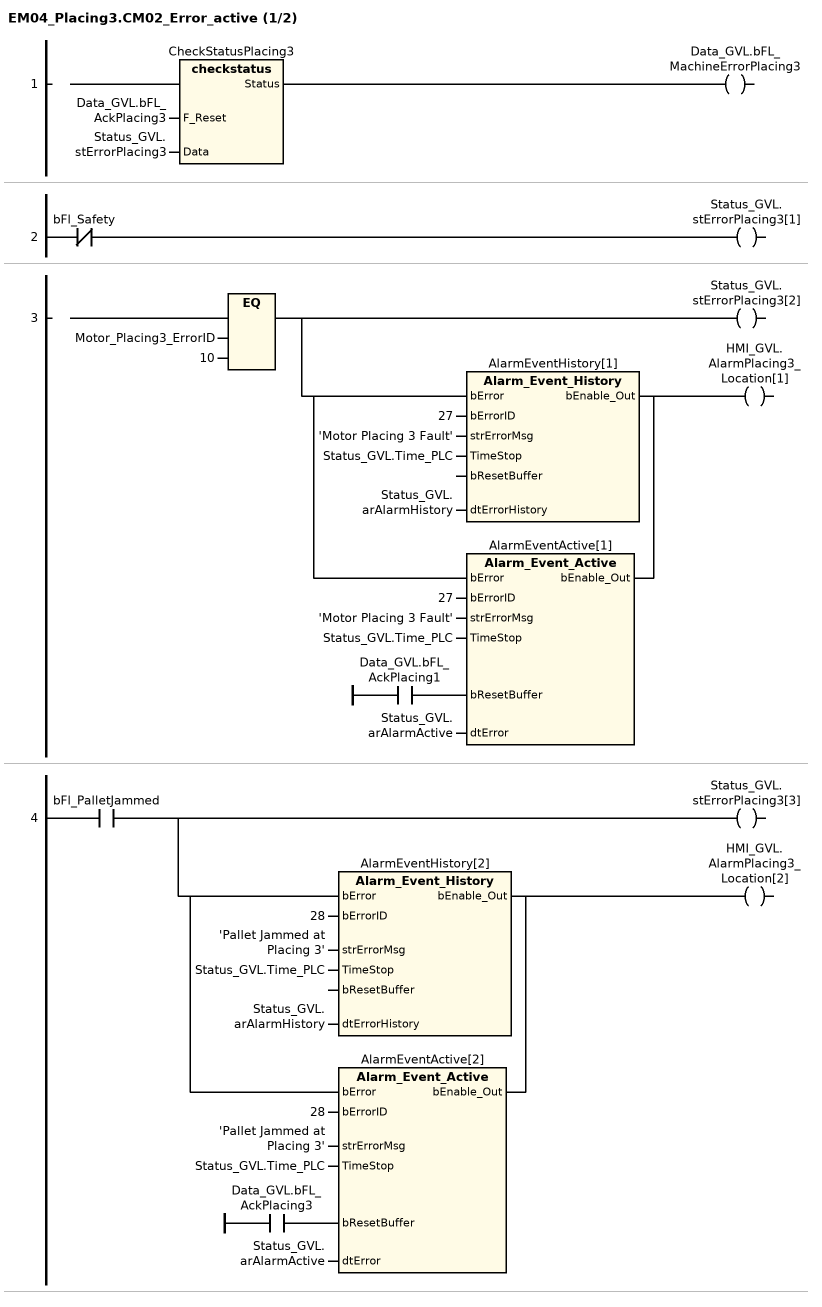
// NETWORK 1
CheckStatusPlacing3(F_Reset := Data_GVL.bFL_AckPlacing3, Data := Status_GVL.stErrorPlacing3); // checkstatus
Data_GVL.bFL_MachineErrorPlacing3 := CheckStatusPlacing3.Status;

// NETWORK 2
Status_GVL.stErrorPlacing3[1] := NOT bFl_Safety;

// NETWORK 3
_w1 := Motor_Placing3_ErrorID = 10;
Status_GVL.stErrorPlacing3[2] := _w1;
AlarmEventHistory[1](
    bError := _w1,
    bErrorID := 27,
    strErrorMsg := 'Motor Placing 3 Fault',
    TimeStop := Status_GVL.Time_PLC,
    dtErrorHistory := Status_GVL.arAlarmHistory); // Alarm_Event_History
AlarmEventActive[1](
    bError := _w1,
    bErrorID := 27,
    strErrorMsg := 'Motor Placing 3 Fault',
    TimeStop := Status_GVL.Time_PLC,
    bResetBuffer := Data_GVL.bFL_AckPlacing1,
    dtError := Status_GVL.arAlarmActive); // Alarm_Event_Active
HMI_GVL.AlarmPlacing3_Location[1] := AlarmEventHistory[1].bEnable_Out OR AlarmEventActive[1].bEnable_Out;

// NETWORK 4
Status_GVL.stErrorPlacing3[3] := bFl_PalletJammed;
AlarmEventHistory[2](
    bError := bFl_PalletJammed,
    bErrorID := 28,
    strErrorMsg := 'Pallet Jammed at Placing 3',
    TimeStop := Status_GVL.Time_PLC,
    dtErrorHistory := Status_GVL.arAlarmHistory); // Alarm_Event_History
AlarmEventActive[2](
    bError := bFl_PalletJammed,
    bErrorID := 28,
    strErrorMsg := 'Pallet Jammed at Placing 3',
    TimeStop := Status_GVL.Time_PLC,
    bResetBuffer := Data_GVL.bFL_AckPlacing3,
    dtError := Status_GVL.arAlarmActive); // Alarm_Event_Active
HMI_GVL.AlarmPlacing3_Location[2] := AlarmEventHistory[2].bEnable_Out OR AlarmEventActive[2].bEnable_Out;

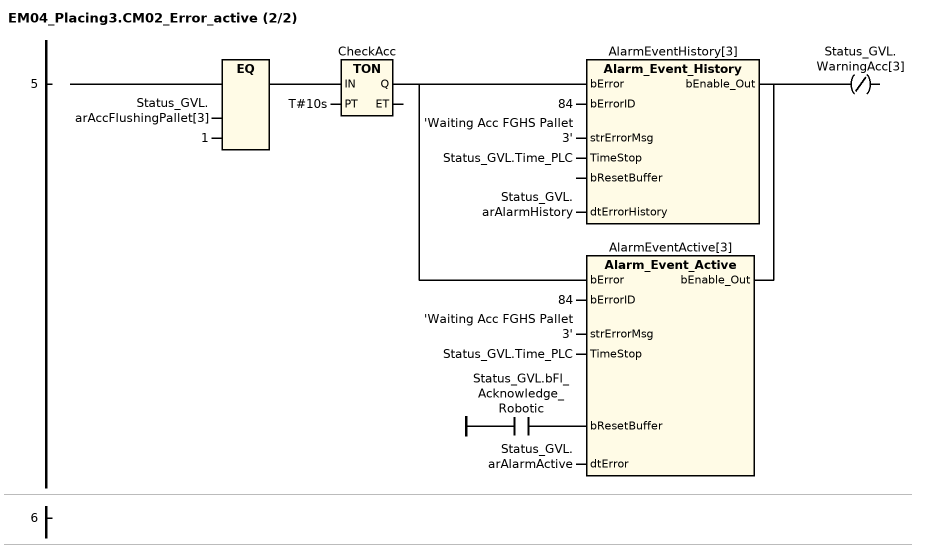
// NETWORK 5
CheckAcc(IN := Status_GVL.arAccFlushingPallet[3] = 1, PT := T#10s); // TON
AlarmEventHistory[3](
    bError := CheckAcc.Q,
    bErrorID := 84,
    strErrorMsg := 'Waiting Acc FGHS Pallet 3',
    TimeStop := Status_GVL.Time_PLC,
    dtErrorHistory := Status_GVL.arAlarmHistory); // Alarm_Event_History
AlarmEventActive[3](
    bError := CheckAcc.Q,
    bErrorID := 84,
    strErrorMsg := 'Waiting Acc FGHS Pallet 3',
    TimeStop := Status_GVL.Time_PLC,
    bResetBuffer := Status_GVL.bFl_Acknowledge_Robotic,
    dtError := Status_GVL.arAlarmActive); // Alarm_Event_Active
Status_GVL.WarningAcc[3] := NOT (AlarmEventHistory[3].bEnable_Out OR AlarmEventActive[3].bEnable_Out);

// NETWORK 6
END_ACTION

ACTION CM03_Output_active:
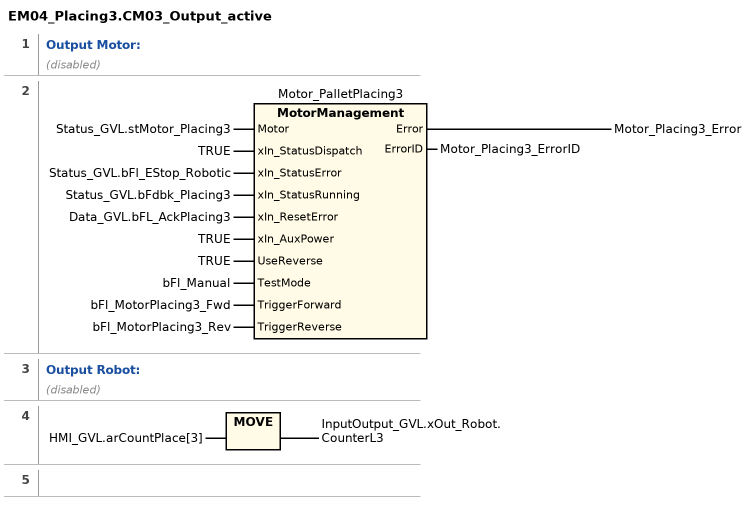
// NETWORK 1 (disabled)
// label: Output Motor

// NETWORK 2
Motor_PalletPlacing3(
    Motor := Status_GVL.stMotor_Placing3,
    xIn_StatusDispatch := TRUE,
    xIn_StatusError := Status_GVL.bFl_EStop_Robotic,
    xIn_StatusRunning := Status_GVL.bFdbk_Placing3,
    xIn_ResetError := Data_GVL.bFL_AckPlacing3,
    xIn_AuxPower := TRUE,
    UseReverse := TRUE,
    TestMode := bFl_Manual,
    TriggerForward := bFl_MotorPlacing3_Fwd,
    TriggerReverse := bFl_MotorPlacing3_Rev,
    ErrorID => Motor_Placing3_ErrorID); // MotorManagement
Motor_Placing3_Error := Motor_PalletPlacing3.Error;

// NETWORK 3 (disabled)
// label: Output Robot

// NETWORK 4
InputOutput_GVL.xOut_Robot.CounterL3 := HMI_GVL.arCountPlace[3];

// NETWORK 5
END_ACTION

ACTION CM04_Running_active:
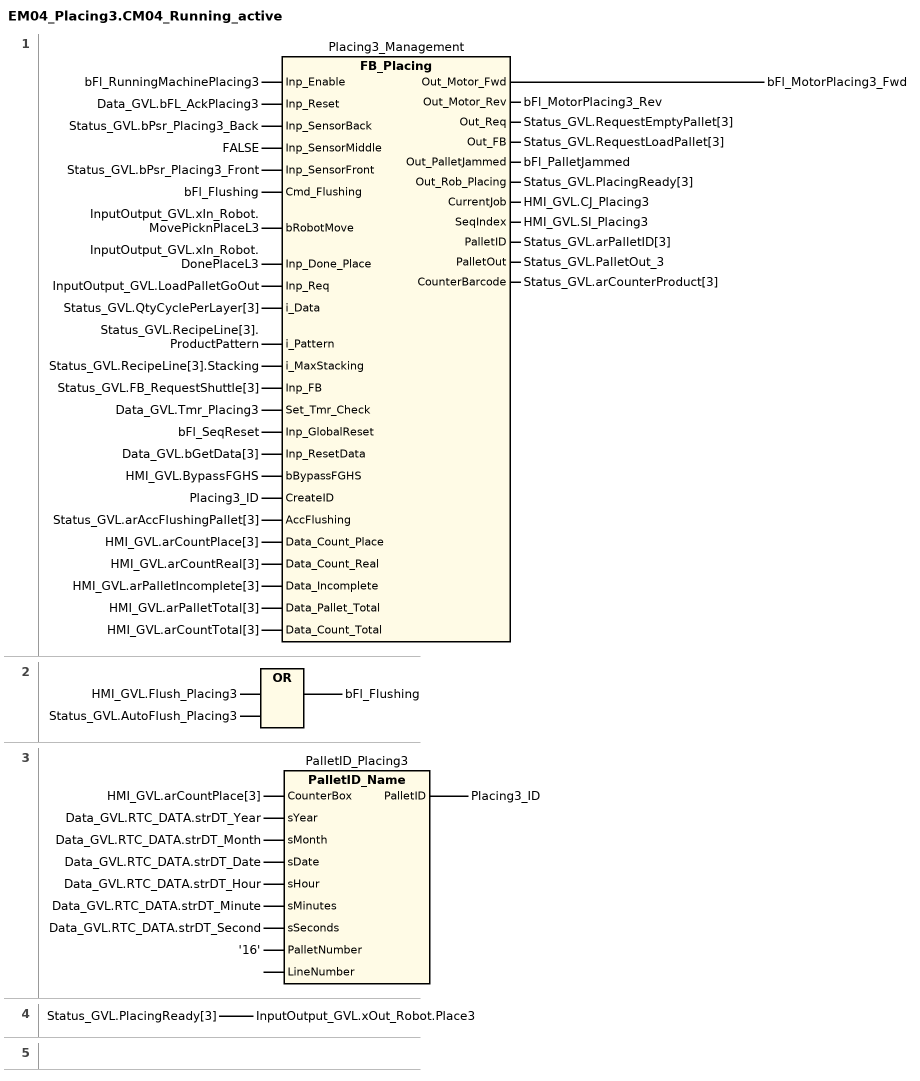
// NETWORK 1
Placing3_Management(
    Inp_Enable := bFl_RunningMachinePlacing3,
    Inp_Reset := Data_GVL.bFL_AckPlacing3,
    Inp_SensorBack := Status_GVL.bPsr_Placing3_Back,
    Inp_SensorMiddle := FALSE,
    Inp_SensorFront := Status_GVL.bPsr_Placing3_Front,
    Cmd_Flushing := bFl_Flushing,
    bRobotMove := InputOutput_GVL.xIn_Robot.MovePicknPlaceL3,
    Inp_Done_Place := InputOutput_GVL.xIn_Robot.DonePlaceL3,
    Inp_Req := InputOutput_GVL.LoadPalletGoOut,
    i_Data := Status_GVL.QtyCyclePerLayer[3],
    i_Pattern := Status_GVL.RecipeLine[3].ProductPattern,
    i_MaxStacking := Status_GVL.RecipeLine[3].Stacking,
    Inp_FB := Status_GVL.FB_RequestShuttle[3],
    Set_Tmr_Check := Data_GVL.Tmr_Placing3,
    Inp_GlobalReset := bFl_SeqReset,
    Inp_ResetData := Data_GVL.bGetData[3],
    bBypassFGHS := HMI_GVL.BypassFGHS,
    CreateID := Placing3_ID,
    AccFlushing := Status_GVL.arAccFlushingPallet[3],
    Data_Count_Place := HMI_GVL.arCountPlace[3],
    Data_Count_Real := HMI_GVL.arCountReal[3],
    Data_Incomplete := HMI_GVL.arPalletIncomplete[3],
    Data_Pallet_Total := HMI_GVL.arPalletTotal[3],
    Data_Count_Total := HMI_GVL.arCountTotal[3],
    Out_Motor_Rev => bFl_MotorPlacing3_Rev,
    Out_Req => Status_GVL.RequestEmptyPallet[3],
    Out_FB => Status_GVL.RequestLoadPallet[3],
    Out_PalletJammed => bFl_PalletJammed,
    Out_Rob_Placing => Status_GVL.PlacingReady[3],
    CurrentJob => HMI_GVL.CJ_Placing3,
    SeqIndex => HMI_GVL.SI_Placing3,
    PalletID => Status_GVL.arPalletID[3],
    PalletOut => Status_GVL.PalletOut_3,
    CounterBarcode => Status_GVL.arCounterProduct[3]); // FB_Placing
bFl_MotorPlacing3_Fwd := Placing3_Management.Out_Motor_Fwd;

// NETWORK 2
bFl_Flushing := HMI_GVL.Flush_Placing3 OR Status_GVL.AutoFlush_Placing3;

// NETWORK 3
PalletID_Placing3(
    CounterBox := HMI_GVL.arCountPlace[3],
    sYear := Data_GVL.RTC_DATA.strDT_Year,
    sMonth := Data_GVL.RTC_DATA.strDT_Month,
    sDate := Data_GVL.RTC_DATA.strDT_Date,
    sHour := Data_GVL.RTC_DATA.strDT_Hour,
    sMinutes := Data_GVL.RTC_DATA.strDT_Minute,
    sSeconds := Data_GVL.RTC_DATA.strDT_Second,
    PalletNumber := '16'); // PalletID_Name
Placing3_ID := PalletID_Placing3.PalletID;

// NETWORK 4
InputOutput_GVL.xOut_Robot.Place3 := Status_GVL.PlacingReady[3];

// NETWORK 5
END_ACTION

ACTION UP01_Backbone_active:
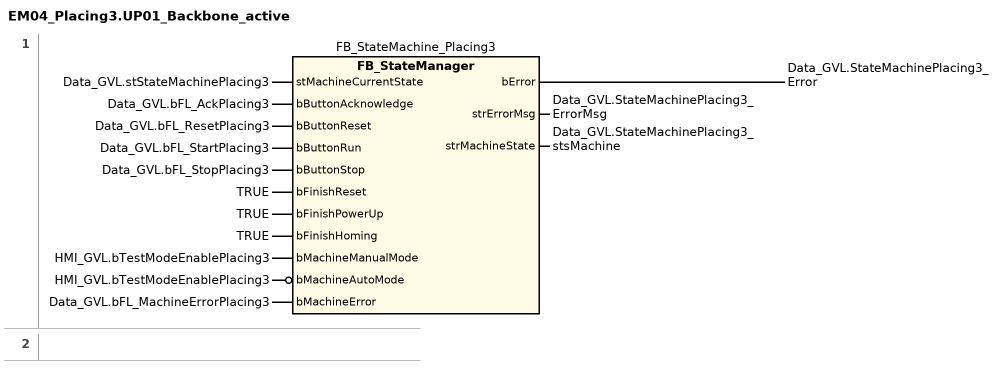
// NETWORK 1
FB_StateMachine_Placing3(
    stMachineCurrentState := Data_GVL.stStateMachinePlacing3,
    bButtonAcknowledge := Data_GVL.bFL_AckPlacing3,
    bButtonReset := Data_GVL.bFL_ResetPlacing3,
    bButtonRun := Data_GVL.bFL_StartPlacing3,
    bButtonStop := Data_GVL.bFL_StopPlacing3,
    bFinishReset := TRUE,
    bFinishPowerUp := TRUE,
    bFinishHoming := TRUE,
    bMachineManualMode := HMI_GVL.bTestModeEnablePlacing3,
    bMachineAutoMode := NOT HMI_GVL.bTestModeEnablePlacing3,
    bMachineError := Data_GVL.bFL_MachineErrorPlacing3,
    strErrorMsg => Data_GVL.StateMachinePlacing3_ErrorMsg,
    strMachineState => Data_GVL.StateMachinePlacing3_stsMachine); // FB_StateManager
Data_GVL.StateMachinePlacing3_Error := FB_StateMachine_Placing3.bError;

// NETWORK 2
END_ACTION

END_PROGRAM

// ---- POUs/S02_Placing/EM05_Placing4.TcPOU
PROGRAM EM05_Placing4
VAR
	
	//Backbone
	FB_StateMachine_Placing4		: FB_StateManager;
	bFl_RunningMachinePlacing4		: BOOL;
	bFl_SeqReset					: BOOL;
	bFl_Manual						: BOOL;
	CheckStatusPlacing4				: checkstatus;
	AlarmEventHistory				: ARRAY[1..20] OF Alarm_Event_History;
	Placing4_Management				: FB_Placing_v2;
	bFl_Flushing					: BOOL;
	PalletID_Placing4				: PalletID_Name;
	Placing4_ID						: STRING;
	bFl_PalletJammed				: BOOL;
	
	//Motor
	Motor_PalletPlacing4			: MotorManagement;
	bFl_MotorPlacing4				: BOOL;
	Motor_Placing4_Error			: BOOL;
	Motor_Placing4_ErrorID			: UINT;
	bFl_MotorPlacing4_Fwd			: BOOL;
	bFl_MotorPlacing4_Rev			: BOOL;
	bFL_Safety						: BOOL;
	AlarmEventActive				: ARRAY[1..20] OF Alarm_Event_Active;
	CheckAcc						: TON;
END_VAR
VAR // added by the converter: edge detectors and wires of the graphical bodies
    _w1 : BOOL;
END_VAR

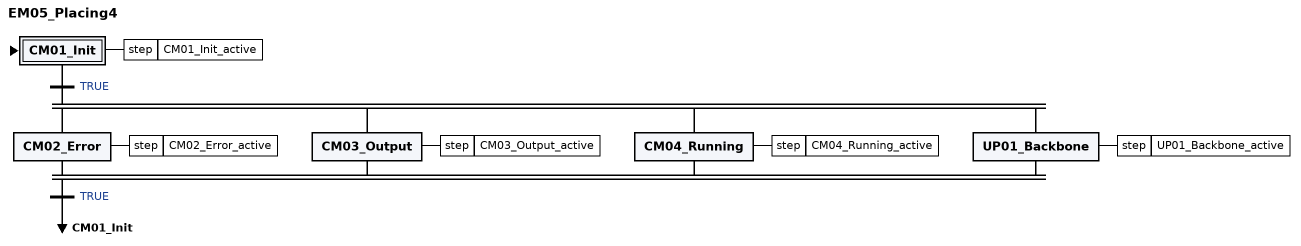
INITIAL_STEP CM01_Init:
    CM01_Init_active(N);  // step action
END_STEP
TRANSITION FROM CM01_Init TO (CM02_Error, CM03_Output, CM04_Running, UP01_Backbone)
    := TRUE;
END_TRANSITION
STEP CM02_Error:
    CM02_Error_active(N);  // step action
END_STEP
STEP CM03_Output:
    CM03_Output_active(N);  // step action
END_STEP
STEP CM04_Running:
    CM04_Running_active(N);  // step action
END_STEP
STEP UP01_Backbone:
    UP01_Backbone_active(N);  // step action
END_STEP
TRANSITION FROM (CM02_Error, CM03_Output, CM04_Running, UP01_Backbone) TO CM01_Init
    := TRUE;
END_TRANSITION

ACTION CM01_Init_active:
Data_GVL.bFL_StartPlacing4			:= Status_GVL.bFl_RunButton_Robotic OR HMI_GVL.bStartButtonPlacing4;
Data_GVL.bFL_StopPlacing4			:= NOT Status_GVL.bFl_StopButton_Robotic OR HMI_GVL.bStopButtonPlacing4;
Data_GVL.bFL_ResetPlacing4			:= Status_GVL.bFl_ResetButton_Robotic OR HMI_GVL.bResetButtonPlacing4;
Data_GVL.bFL_AckPlacing4			:= Status_GVL.bFl_Acknowledge_Robotic OR HMI_GVL.bAcknowledgeButtonPlacing4;
Data_GVL.bFL_AutoManuaModePlacing4 	:= Status_GVL.bFl_Manual_Robotic OR HMI_GVL.bTestModeEnablePlacing4;
bFl_RunningMachinePlacing4			:= Data_GVL.stStateMachinePlacing4.Running;
bFl_Manual							:= Data_GVL.stStateMachinePlacing4.ManualMode;
bFl_SeqReset						:= NOT Status_GVL.bFl_EStop_Robotic;
bFL_Safety							:= Status_GVL.bFl_EStop_Robotic AND Status_GVL.bSafety_DoorRobotic;



(*=================Convert Timer============================*)
Data_GVL.Tmr_Placing4	:= ConvertMilliSecTimeData(HMI_GVL.Tmr_Placing4);

(*=================Data OEE============================*)
Data_GVL.dt_Production[4].Data1			:= HMI_GVL.arCountTotal[4];
Data_GVL.dt_Production[4].Data2			:= HMI_GVL.arPalletTotal[4];
Data_GVL.dt_Production[4].Data3			:= HMI_GVL.arPalletIncomplete[4];
Data_GVL.dt_Production[4].ProductCode	:= Status_GVL.RecipeLine[4].ProductName;
END_ACTION

ACTION CM02_Error_active:
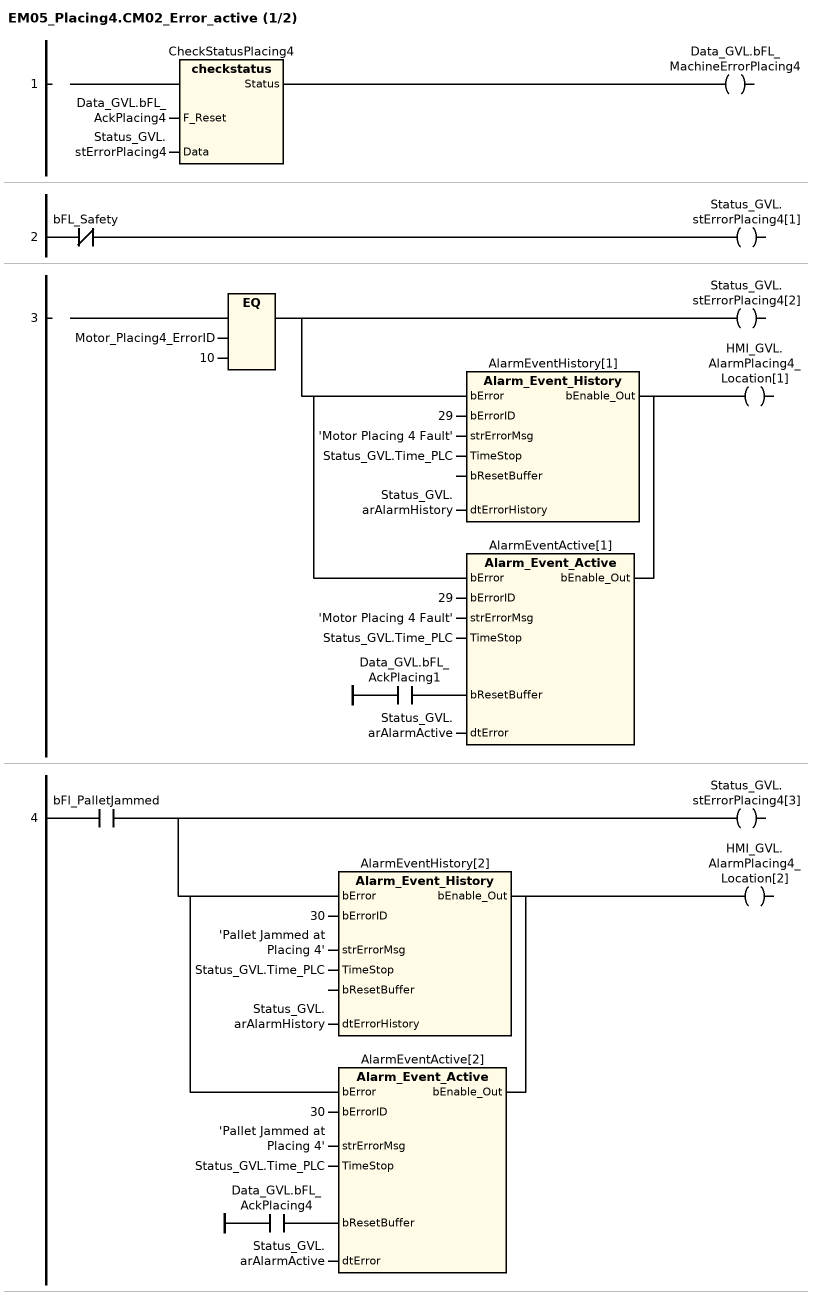
// NETWORK 1
CheckStatusPlacing4(F_Reset := Data_GVL.bFL_AckPlacing4, Data := Status_GVL.stErrorPlacing4); // checkstatus
Data_GVL.bFL_MachineErrorPlacing4 := CheckStatusPlacing4.Status;

// NETWORK 2
Status_GVL.stErrorPlacing4[1] := NOT bFL_Safety;

// NETWORK 3
_w1 := Motor_Placing4_ErrorID = 10;
Status_GVL.stErrorPlacing4[2] := _w1;
AlarmEventHistory[1](
    bError := _w1,
    bErrorID := 29,
    strErrorMsg := 'Motor Placing 4 Fault',
    TimeStop := Status_GVL.Time_PLC,
    dtErrorHistory := Status_GVL.arAlarmHistory); // Alarm_Event_History
AlarmEventActive[1](
    bError := _w1,
    bErrorID := 29,
    strErrorMsg := 'Motor Placing 4 Fault',
    TimeStop := Status_GVL.Time_PLC,
    bResetBuffer := Data_GVL.bFL_AckPlacing1,
    dtError := Status_GVL.arAlarmActive); // Alarm_Event_Active
HMI_GVL.AlarmPlacing4_Location[1] := AlarmEventHistory[1].bEnable_Out OR AlarmEventActive[1].bEnable_Out;

// NETWORK 4
Status_GVL.stErrorPlacing4[3] := bFl_PalletJammed;
AlarmEventHistory[2](
    bError := bFl_PalletJammed,
    bErrorID := 30,
    strErrorMsg := 'Pallet Jammed at Placing 4',
    TimeStop := Status_GVL.Time_PLC,
    dtErrorHistory := Status_GVL.arAlarmHistory); // Alarm_Event_History
AlarmEventActive[2](
    bError := bFl_PalletJammed,
    bErrorID := 30,
    strErrorMsg := 'Pallet Jammed at Placing 4',
    TimeStop := Status_GVL.Time_PLC,
    bResetBuffer := Data_GVL.bFL_AckPlacing4,
    dtError := Status_GVL.arAlarmActive); // Alarm_Event_Active
HMI_GVL.AlarmPlacing4_Location[2] := AlarmEventHistory[2].bEnable_Out OR AlarmEventActive[2].bEnable_Out;

